C09147=1141.971,319.526,-76.453,-176.806,8.868,148.842
C09148=1141.967,319.774,-76.485,-176.803,8.872,148.842
C09149=1141.963,320.022,-76.518,-176.800,8.876,148.843
C09150=1141.958,320.270,-76.550,-176.798,8.880,148.843
C09151=1141.954,320.517,-76.583,-176.795,8.883,148.843
C09152=1141.950,320.766,-76.615,-176.792,8.887,148.843
C09153=1141.946,321.013,-76.648,-176.790,8.890,148.843
C09154=1141.942,321.261,-76.680,-176.787,8.894,148.844
C09155=1141.938,321.509,-76.713,-176.785,8.898,148.844
C09156=1141.934,321.757,-76.745,-176.782,8.902,148.844
C09157=1141.930,322.005,-76.778,-176.779,8.905,148.844
C09158=1141.926,322.253,-76.810,-176.776,8.909,148.844
C09159=1141.922,322.501,-76.843,-176.774,8.912,148.845
C09160=1141.917,322.748,-76.876,-176.771,8.916,148.845
C09161=1141.914,322.996,-76.908,-176.769,8.920,148.845
C09162=1141.910,323.243,-76.941,-176.766,8.924,148.845
C09163=1141.905,323.492,-76.973,-176.764,8.927,148.845
C09164=1141.901,323.739,-77.006,-176.761,8.931,148.846
C09165=1141.898,323.987,-77.039,-176.758,8.934,148.846
C09166=1141.893,324.235,-77.071,-176.756,8.938,148.846
C09167=1141.889,324.483,-77.105,-176.753,8.942,148.846
C09168=1141.886,324.730,-77.137,-176.751,8.945,148.847
C09169=1141.881,324.978,-77.170,-176.748,8.949,148.847
C09170=1141.877,325.226,-77.203,-176.746,8.953,148.847
C09171=1141.873,325.474,-77.236,-176.743,8.957,148.847
C09172=1141.869,325.722,-77.269,-176.741,8.960,148.848
C09173=1141.865,325.969,-77.302,-176.738,8.964,148.848
C09174=1141.861,326.218,-77.334,-176.735,8.967,148.848
C09175=1141.857,326.465,-77.367,-176.732,8.971,148.848
C09176=1141.853,326.713,-77.400,-176.730,8.975,148.848
C09177=1141.848,326.961,-77.434,-176.727,8.979,148.849
C09178=1141.844,327.209,-77.467,-176.724,8.983,148.849
C09179=1141.841,327.456,-77.499,-176.722,8.986,148.849
C09180=1141.836,327.704,-77.532,-176.719,8.990,148.849
C09181=1141.832,327.952,-77.565,-176.717,8.994,148.850
C09182=1141.828,328.200,-77.598,-176.714,8.998,148.850
C09183=1141.824,328.448,-77.631,-176.712,9.001,148.850
C09184=1141.820,328.695,-77.664,-176.709,9.005,148.850
C09185=1141.816,328.943,-77.698,-176.707,9.008,148.851
C09186=1141.812,329.191,-77.731,-176.704,9.012,148.851
C09187=1141.807,329.438,-77.764,-176.702,9.016,148.851
C09188=1141.804,329.687,-77.797,-176.699,9.020,148.851
C09189=1141.801,329.934,-77.830,-176.697,9.023,148.852
C09190=1141.796,330.182,-77.863,-176.694,9.027,148.852
C09191=1141.792,330.430,-77.896,-176.691,9.031,148.852
C09192=1141.788,330.677,-77.929,-176.688,9.035,148.852
C09193=1141.784,330.925,-77.963,-176.686,9.038,148.853
C09194=1141.780,331.173,-77.996,-176.683,9.042,148.853
C09195=1141.776,331.421,-78.029,-176.681,9.047,148.853
C09196=1141.772,331.668,-78.063,-176.678,9.050,148.853
C09197=1141.768,331.915,-78.096,-176.675,9.054,148.854
C09198=1141.764,332.164,-78.129,-176.673,9.057,148.854
C09199=1141.760,332.412,-78.163,-176.670,9.062,148.854
C09200=1141.755,332.660,-78.196,-176.668,9.065,148.854
C09201=1141.751,332.907,-78.229,-176.665,9.069,148.855
C09202=1141.747,333.155,-78.263,-176.663,9.072,148.855
C09203=1141.743,333.402,-78.296,-176.660,9.077,148.855
C09204=1141.739,333.650,-78.330,-176.657,9.081,148.856
C09205=1141.735,333.898,-78.363,-176.655,9.084,148.856
C09206=1141.732,334.146,-78.397,-176.652,9.088,148.856
C09207=1141.727,334.393,-78.430,-176.650,9.092,148.856
C09208=1141.723,334.641,-78.463,-176.647,9.096,148.857
C09209=1141.719,334.889,-78.497,-176.645,9.099,148.857
C09210=1141.716,335.137,-78.531,-176.642,9.103,148.857
C09211=1141.711,335.385,-78.564,-176.640,9.106,148.857
C09212=1141.707,335.632,-78.598,-176.637,9.111,148.858
C09213=1141.703,335.879,-78.632,-176.634,9.115,148.858
C09214=1141.699,336.127,-78.665,-176.632,9.118,148.858
C09215=1141.696,336.375,-78.699,-176.629,9.122,148.859
C09216=1141.691,336.623,-78.733,-176.627,9.126,148.859
C09217=1141.687,336.871,-78.766,-176.624,9.130,148.859
C09218=1141.683,337.118,-78.800,-176.621,9.134,148.859
C09219=1141.679,337.366,-78.833,-176.619,9.137,148.860
C09220=1141.676,337.613,-78.867,-176.616,9.141,148.860
C09221=1141.671,337.861,-78.901,-176.614,9.145,148.860
C09222=1141.667,338.109,-78.935,-176.612,9.149,148.860
C09223=1141.663,338.357,-78.968,-176.609,9.152,148.861
C09224=1141.659,338.604,-79.002,-176.606,9.156,148.861
C09225=1141.655,338.885,-79.041,-176.604,9.161,148.861
C09226=1141.650,339.165,-79.079,-176.601,9.165,148.862
C09227=1141.645,339.446,-79.118,-176.597,9.170,148.862
C09228=1141.641,339.726,-79.155,-176.595,9.174,148.862
C09229=1141.636,339.974,-79.189,-176.593,9.177,148.863
C09230=1141.633,340.222,-79.223,-176.590,9.181,148.863
C09231=1141.629,340.469,-79.257,-176.587,9.186,148.863
C09232=1141.624,340.717,-79.291,-176.585,9.189,148.863
C09233=1141.621,340.965,-79.325,-176.582,9.193,148.864
C09234=1141.617,341.212,-79.360,-176.579,9.198,148.864
C09235=1141.612,341.460,-79.393,-176.577,9.201,148.864
C09236=1141.609,341.708,-79.427,-176.574,9.205,148.865
C09237=1141.605,341.955,-79.462,-176.572,9.208,148.865
C09238=1141.601,342.203,-79.495,-176.569,9.213,148.865
C09239=1141.597,342.451,-79.530,-176.566,9.217,148.865
C09240=1141.593,342.698,-79.564,-176.564,9.220,148.866
C09241=1141.588,342.946,-79.598,-176.562,9.224,148.866
C09242=1141.585,343.194,-79.632,-176.559,9.229,148.867
C09243=1141.581,343.441,-79.665,-176.557,9.232,148.867
C09244=1141.576,343.689,-79.700,-176.554,9.236,148.867
C09245=1141.573,343.937,-79.734,-176.552,9.240,148.867
C09246=1141.568,344.184,-79.769,-176.549,9.244,148.868
C09247=1141.565,344.432,-79.803,-176.546,9.248,148.868
C09248=1141.561,344.679,-79.837,-176.544,9.251,148.868
C09249=1141.557,344.926,-79.871,-176.541,9.255,148.869
C09250=1141.553,345.174,-79.906,-176.539,9.260,148.869
C09251=1141.549,345.421,-79.940,-176.536,9.263,148.869
C09252=1141.545,345.670,-79.974,-176.534,9.267,148.870
C09253=1141.540,345.918,-80.008,-176.531,9.271,148.870
C09254=1141.537,346.165,-80.043,-176.529,9.275,148.870
C09255=1141.532,346.413,-80.077,-176.526,9.279,148.871
C09256=1141.529,346.660,-80.111,-176.524,9.282,148.871
C09257=1141.525,346.908,-80.146,-176.521,9.287,148.871
C09258=1141.521,347.155,-80.180,-176.518,9.291,148.871
C09259=1141.517,347.403,-80.215,-176.516,9.294,148.872
C09260=1141.512,347.650,-80.250,-176.513,9.299,148.872
C09261=1141.509,347.898,-80.284,-176.511,9.303,148.873
C09262=1141.505,348.145,-80.318,-176.509,9.306,148.873
C09263=1141.501,348.393,-80.353,-176.506,9.311,148.873
C09264=1141.497,348.641,-80.387,-176.503,9.315,148.873
C09265=1141.493,348.889,-80.422,-176.501,9.318,148.874
C09266=1141.489,349.136,-80.456,-176.498,9.322,148.874
C09267=1141.485,349.383,-80.491,-176.496,9.327,148.875
C09268=1141.481,349.631,-80.526,-176.494,9.330,148.875
C09269=1141.478,349.879,-80.560,-176.491,9.334,148.875
C09270=1141.473,350.126,-80.595,-176.488,9.338,148.876
C09271=1141.469,350.374,-80.629,-176.486,9.342,148.876
C09272=1141.465,350.621,-80.665,-176.483,9.346,148.876
C09273=1141.462,350.869,-80.699,-176.481,9.350,148.877
C09274=1141.458,351.117,-80.734,-176.478,9.354,148.877
C09275=1141.453,351.364,-80.769,-176.476,9.358,148.877
C09276=1141.449,351.612,-80.804,-176.473,9.362,148.878
C09277=1141.446,351.859,-80.837,-176.470,9.367,148.878
C09278=1141.442,352.106,-80.873,-176.468,9.370,148.878
C09279=1141.437,352.354,-80.908,-176.466,9.374,148.879
C09280=1141.433,352.602,-80.942,-176.463,9.378,148.879
C09281=1141.430,352.849,-80.977,-176.461,9.382,148.879
C09282=1141.426,353.097,-81.012,-176.458,9.386,148.880
C09283=1141.422,353.344,-81.047,-176.455,9.390,148.880
C09284=1141.418,353.591,-81.082,-176.453,9.394,148.880
C09285=1141.414,353.840,-81.117,-176.451,9.398,148.881
C09286=1141.410,354.087,-81.152,-176.448,9.402,148.881
C09287=1141.406,354.334,-81.186,-176.446,9.406,148.881
C09288=1141.402,354.582,-81.222,-176.443,9.410,148.882
C09289=1141.399,354.830,-81.256,-176.440,9.414,148.882
C09290=1141.394,355.077,-81.292,-176.438,9.418,148.882
C09291=1141.390,355.325,-81.326,-176.435,9.422,148.883
C09292=1141.387,355.572,-81.362,-176.433,9.426,148.883
C09293=1141.382,355.819,-81.397,-176.430,9.430,148.884
C09294=1141.378,356.067,-81.432,-176.428,9.434,148.884
C09295=1141.375,356.315,-81.468,-176.426,9.438,148.884
C09296=1141.371,356.562,-81.501,-176.423,9.442,148.885
C09297=1141.367,356.809,-81.537,-176.420,9.447,148.885
C09298=1141.364,357.057,-81.572,-176.418,9.450,148.885
C09299=1141.359,357.304,-81.607,-176.415,9.454,148.886
C09300=1141.355,357.552,-81.643,-176.413,9.459,148.886
C09301=1141.352,357.799,-81.678,-176.410,9.463,148.886
C09302=1141.347,358.047,-81.713,-176.408,9.466,148.887
C09303=1141.343,358.294,-81.748,-176.405,9.471,148.887
C09304=1141.340,358.542,-81.784,-176.402,9.475,148.887
C09305=1141.336,358.789,-81.819,-176.400,9.479,148.888
C09306=1141.332,359.037,-81.854,-176.398,9.483,148.888
C09307=1141.328,359.284,-81.889,-176.395,9.487,148.889
C09308=1141.324,359.532,-81.925,-176.393,9.491,148.889
C09309=1141.321,359.779,-81.960,-176.390,9.495,148.889
C09310=1141.316,360.026,-81.995,-176.388,9.499,148.890
C09311=1141.313,360.273,-82.031,-176.385,9.503,148.890
C09312=1141.309,360.521,-82.066,-176.382,9.507,148.890
C09313=1141.304,360.769,-82.102,-176.380,9.512,148.891
C09314=1141.301,361.017,-82.138,-176.377,9.516,148.891
C09315=1141.296,361.264,-82.173,-176.374,9.520,148.892
C09316=1141.293,361.511,-82.208,-176.372,9.524,148.892
C09317=1141.289,361.759,-82.244,-176.370,9.528,148.892
C09318=1141.285,362.006,-82.279,-176.367,9.532,148.893
C09319=1141.282,362.254,-82.315,-176.365,9.537,148.893
C09320=1141.277,362.500,-82.350,-176.362,9.541,148.893
C09321=1141.274,362.748,-82.386,-176.359,9.545,148.894
C09322=1141.269,362.996,-82.422,-176.356,9.549,148.894
C09323=1141.266,363.243,-82.457,-176.354,9.553,148.895
C09324=1141.262,363.491,-82.493,-176.352,9.557,148.895
C09325=1141.258,363.738,-82.528,-176.349,9.561,148.895
C09326=1141.255,363.986,-82.564,-176.346,9.565,148.896
C09327=1141.250,364.233,-82.600,-176.344,9.570,148.896
C09328=1141.246,364.480,-82.635,-176.341,9.574,148.897
C09329=1141.242,364.764,-82.676,-176.338,9.579,148.897
C09330=1141.238,365.048,-82.717,-176.335,9.583,148.898
C09331=1141.233,365.331,-82.759,-176.332,9.588,148.898
C09332=1141.229,365.616,-82.800,-176.329,9.594,148.898
C09333=1141.225,365.863,-82.835,-176.326,9.598,148.899
C09334=1141.221,366.109,-82.871,-176.323,9.602,148.899
C09335=1141.217,366.357,-82.907,-176.321,9.606,148.900
C09336=1141.213,366.604,-82.943,-176.319,9.610,148.900
C09337=1141.209,366.852,-82.978,-176.316,9.614,148.900
C09338=1141.205,367.099,-83.015,-176.313,9.618,148.901
C09339=1141.202,367.347,-83.051,-176.311,9.623,148.901
C09340=1141.198,367.594,-83.086,-176.308,9.627,148.901
C09341=1141.194,367.841,-83.123,-176.305,9.631,148.902
C09342=1141.190,368.089,-83.159,-176.303,9.636,148.902
C09343=1141.186,368.337,-83.195,-176.300,9.640,148.903
C09344=1141.183,368.584,-83.231,-176.297,9.644,148.903
C09345=1141.179,368.831,-83.267,-176.295,9.649,148.904
C09346=1141.174,369.079,-83.303,-176.292,9.653,148.904
C09347=1141.171,369.326,-83.339,-176.289,9.657,148.904
C09348=1141.167,369.574,-83.375,-176.287,9.661,148.905
C09349=1141.163,369.820,-83.412,-176.284,9.665,148.905
C09350=1141.160,370.068,-83.447,-176.281,9.670,148.905
C09351=1141.156,370.315,-83.484,-176.279,9.674,148.906
C09352=1141.152,370.563,-83.520,-176.276,9.678,148.906
C09353=1141.148,370.810,-83.556,-176.273,9.683,148.907
C09354=1141.144,371.057,-83.592,-176.271,9.687,148.907
C09355=1141.140,371.305,-83.629,-176.268,9.691,148.908
C09356=1141.136,371.552,-83.664,-176.266,9.695,148.908
C09357=1141.132,371.799,-83.701,-176.263,9.700,148.908
C09358=1141.129,372.046,-83.737,-176.261,9.704,148.909
C09359=1141.125,372.294,-83.774,-176.259,9.708,148.909
C09360=1141.121,372.541,-83.810,-176.256,9.712,148.910
C09361=1141.117,372.789,-83.846,-176.253,9.716,148.910
C09362=1141.113,373.036,-83.883,-176.251,9.721,148.910
C09363=1141.109,373.283,-83.919,-176.248,9.725,148.911
C09364=1141.105,373.530,-83.955,-176.246,9.729,148.911
C09365=1141.102,373.777,-83.992,-176.243,9.734,148.912
C09366=1141.098,374.025,-84.029,-176.241,9.737,148.912
C09367=1141.095,374.272,-84.065,-176.239,9.742,148.913
C09368=1141.090,374.520,-84.101,-176.236,9.746,148.913
C09369=1141.086,374.767,-84.138,-176.233,9.750,148.913
C09370=1141.083,375.014,-84.174,-176.231,9.754,148.914
C09371=1141.079,375.261,-84.211,-176.229,9.758,148.914
C09372=1141.075,375.508,-84.248,-176.226,9.763,148.915
C09373=1141.071,375.756,-84.284,-176.224,9.766,148.915
C09374=1141.067,376.003,-84.320,-176.222,9.770,148.916
C09375=1141.063,376.251,-84.358,-176.220,9.775,148.916
C09376=1141.060,376.498,-84.394,-176.218,9.779,148.917
C09377=1141.056,376.745,-84.431,-176.215,9.783,148.917
C09378=1141.052,376.992,-84.468,-176.213,9.787,148.918
C09379=1141.049,377.239,-84.504,-176.211,9.791,148.918
C09380=1141.044,377.486,-84.541,-176.209,9.795,148.919
C09381=1141.041,377.734,-84.578,-176.206,9.799,148.919
C09382=1141.037,377.982,-84.614,-176.205,9.803,148.920
C09383=1141.033,378.229,-84.650,-176.203,9.806,148.920
C09384=1141.029,378.476,-84.687,-176.200,9.811,148.920
C09385=1141.025,378.723,-84.724,-176.199,9.815,148.921
C09386=1141.021,378.970,-84.761,-176.197,9.818,148.921
C09387=1141.018,379.218,-84.798,-176.195,9.822,148.922
C09388=1141.014,379.465,-84.834,-176.194,9.826,148.923
C09389=1141.010,379.712,-84.872,-176.191,9.830,148.923
C09390=1141.006,379.959,-84.909,-176.189,9.834,148.924
C09391=1141.002,380.206,-84.946,-176.188,9.838,148.924
C09392=1140.999,380.454,-84.982,-176.186,9.841,148.925
C09393=1140.995,380.701,-85.019,-176.185,9.845,148.925
C09394=1140.991,380.948,-85.056,-176.183,9.848,148.926
C09395=1140.987,381.195,-85.093,-176.182,9.852,148.926
C09396=1140.984,381.443,-85.130,-176.180,9.856,148.927
C09397=1140.979,381.690,-85.167,-176.179,9.860,148.927
C09398=1140.976,381.937,-85.203,-176.177,9.862,148.928
C09399=1140.972,382.184,-85.241,-176.176,9.866,148.928
C09400=1140.969,382.432,-85.278,-176.175,9.869,148.929
C09401=1140.965,382.679,-85.315,-176.173,9.873,148.930
C09402=1140.961,382.926,-85.352,-176.172,9.876,148.930
C09403=1140.957,383.173,-85.389,-176.171,9.880,148.931
C09404=1140.953,383.421,-85.427,-176.170,9.884,148.931
C09405=1140.949,383.668,-85.463,-176.170,9.887,148.932
C09406=1140.945,383.915,-85.500,-176.169,9.890,148.933
C09407=1140.942,384.162,-85.537,-176.168,9.893,148.933
C09408=1140.939,384.409,-85.574,-176.167,9.896,148.934
C09409=1140.935,384.656,-85.611,-176.166,9.899,148.934
C09410=1140.930,384.904,-85.648,-176.166,9.903,148.935
C09411=1140.927,385.151,-85.685,-176.165,9.906,148.936
C09412=1140.923,385.398,-85.723,-176.165,9.908,148.936
C09413=1140.919,385.645,-85.760,-176.164,9.911,148.937
C09414=1140.916,385.893,-85.797,-176.164,9.915,148.938
C09415=1140.912,386.140,-85.834,-176.164,9.917,148.938
C09416=1140.908,386.387,-85.872,-176.163,9.921,148.939
C09417=1140.904,386.634,-85.908,-176.163,9.923,148.940
C09418=1140.900,386.882,-85.946,-176.163,9.925,148.940
C09419=1140.896,387.128,-85.983,-176.162,9.929,148.941
C09420=1140.892,387.376,-86.020,-176.162,9.931,148.942
C09421=1140.889,387.624,-86.057,-176.163,9.934,148.943
C09422=1140.886,387.870,-86.094,-176.163,9.936,148.943
C09423=1140.882,388.117,-86.131,-176.163,9.939,148.944
C09424=1140.878,388.365,-86.168,-176.163,9.942,148.945
C09425=1140.874,388.611,-86.206,-176.163,9.944,148.946
C09426=1140.870,388.859,-86.243,-176.163,9.947,148.946
C09427=1140.867,389.107,-86.280,-176.163,9.950,148.947
C09428=1140.863,389.353,-86.318,-176.164,9.952,148.948
C09429=1140.859,389.600,-86.354,-176.164,9.955,148.949
C09430=1140.856,389.848,-86.392,-176.165,9.957,148.949
C09431=1140.852,390.095,-86.429,-176.165,9.960,148.950
C09432=1140.847,390.342,-86.466,-176.165,9.962,148.951
C09433=1140.843,390.629,-86.510,-176.166,9.964,148.952
C09434=1140.839,390.917,-86.553,-176.167,9.967,148.952
C09435=1140.834,391.204,-86.596,-176.167,9.970,148.953
C09436=1140.830,391.491,-86.640,-176.168,9.973,148.954
C09437=1140.826,391.738,-86.677,-176.169,9.975,148.955
C09438=1140.823,391.985,-86.715,-176.169,9.978,148.956
C09439=1140.819,392.233,-86.751,-176.170,9.980,148.957
C09440=1140.815,392.480,-86.788,-176.171,9.982,148.957
C09441=1140.811,392.727,-86.826,-176.172,9.984,148.958
C09442=1140.807,392.974,-86.863,-176.173,9.987,148.959
C09443=1140.804,393.221,-86.901,-176.174,9.988,148.960
C09444=1140.800,393.469,-86.938,-176.174,9.991,148.961
C09445=1140.796,393.716,-86.975,-176.175,9.993,148.962
C09446=1140.792,393.962,-87.012,-176.176,9.995,148.962
C09447=1140.789,394.210,-87.050,-176.177,9.997,148.963
C09448=1140.785,394.457,-87.087,-176.178,9.999,148.964
C09449=1140.781,394.704,-87.124,-176.179,10.001,148.965
C09450=1140.777,394.952,-87.161,-176.180,10.004,148.966
C09451=1140.773,395.198,-87.199,-176.181,10.006,148.966
C09452=1140.769,395.446,-87.236,-176.182,10.008,148.967
C09453=1140.766,395.693,-87.274,-176.183,10.010,148.968
C09454=1140.762,395.940,-87.310,-176.184,10.012,148.969
C09455=1140.758,396.187,-87.347,-176.185,10.014,148.970
C09456=1140.755,396.435,-87.385,-176.186,10.016,148.971
C09457=1140.751,396.682,-87.422,-176.187,10.018,148.971
C09458=1140.747,396.928,-87.460,-176.188,10.021,148.972
C09459=1140.743,397.176,-87.497,-176.189,10.023,148.973
C09460=1140.739,397.423,-87.534,-176.190,10.025,148.974
C09461=1140.736,397.670,-87.571,-176.192,10.027,148.975
C09462=1140.732,397.918,-87.609,-176.193,10.029,148.976
C09463=1140.728,398.164,-87.646,-176.194,10.031,148.976
C09464=1140.724,398.412,-87.683,-176.195,10.032,148.977
C09465=1140.721,398.659,-87.721,-176.197,10.034,148.978
C09466=1140.717,398.906,-87.758,-176.198,10.037,148.979
C09467=1140.713,399.153,-87.795,-176.199,10.039,148.980
C09468=1140.710,399.401,-87.833,-176.200,10.041,148.981
C09469=1140.706,399.648,-87.869,-176.201,10.043,148.981
C09470=1140.702,399.894,-87.907,-176.202,10.045,148.982
C09471=1140.698,400.142,-87.944,-176.203,10.047,148.983
C09472=1140.694,400.389,-87.981,-176.205,10.048,148.984
C09473=1140.690,400.636,-88.019,-176.206,10.050,148.985
C09474=1140.687,400.884,-88.056,-176.208,10.053,148.986
C09475=1140.683,401.130,-88.093,-176.209,10.055,148.987
C09476=1140.679,401.378,-88.130,-176.210,10.057,148.987
C09477=1140.675,401.626,-88.168,-176.211,10.059,148.988
C09478=1140.672,401.872,-88.205,-176.212,10.061,148.989
C09479=1140.668,402.119,-88.242,-176.214,10.062,148.990
C09480=1140.664,402.367,-88.280,-176.215,10.064,148.991
C09481=1140.660,402.614,-88.317,-176.216,10.066,148.992
C09482=1140.656,402.861,-88.354,-176.217,10.069,148.993
C09483=1140.653,403.108,-88.392,-176.218,10.071,148.993
C09484=1140.649,403.355,-88.428,-176.219,10.073,148.994
C09485=1140.645,403.602,-88.466,-176.221,10.075,148.995
C09486=1140.642,403.850,-88.503,-176.222,10.076,148.996
C09487=1140.638,404.097,-88.540,-176.223,10.078,148.997
C09488=1140.634,404.344,-88.578,-176.225,10.080,148.998
C09489=1140.630,404.592,-88.615,-176.226,10.082,148.999
C09490=1140.627,404.838,-88.652,-176.227,10.085,148.999
C09491=1140.622,405.086,-88.690,-176.228,10.087,149.000
C09492=1140.618,405.333,-88.728,-176.229,10.089,149.001
C09493=1140.614,405.580,-88.765,-176.230,10.091,149.002
C09494=1140.610,405.827,-88.802,-176.231,10.093,149.003
C09495=1140.607,406.075,-88.840,-176.233,10.094,149.003
C09496=1140.603,406.322,-88.876,-176.234,10.096,149.004
C09497=1140.599,406.568,-88.914,-176.235,10.098,149.005
C09498=1140.596,406.816,-88.951,-176.237,10.101,149.006
C09499=1140.592,407.063,-88.988,-176.238,10.103,149.007
C09500=1140.588,407.310,-89.026,-176.239,10.105,149.008
C09501=1140.584,407.558,-89.063,-176.240,10.107,149.009
C09502=1140.581,407.804,-89.100,-176.241,10.109,149.009
C09503=1140.576,408.052,-89.137,-176.242,10.111,149.010
C09504=1140.573,408.299,-89.174,-176.243,10.113,149.011
C09505=1140.569,408.546,-89.212,-176.244,10.115,149.012
C09506=1140.565,408.793,-89.249,-176.245,10.117,149.013
C09507=1140.562,409.041,-89.287,-176.246,10.119,149.014
C09508=1140.558,409.288,-89.324,-176.247,10.121,149.014
C09509=1140.554,409.535,-89.361,-176.249,10.123,149.015
C09510=1140.551,409.782,-89.399,-176.250,10.125,149.016
C09511=1140.546,410.029,-89.435,-176.251,10.127,149.017
C09512=1140.543,410.276,-89.473,-176.252,10.129,149.018
C09513=1140.539,410.524,-89.510,-176.253,10.132,149.019
C09514=1140.535,410.771,-89.547,-176.254,10.134,149.019
C09515=1140.531,411.018,-89.585,-176.255,10.135,149.020
C09516=1140.528,411.265,-89.622,-176.255,10.138,149.021
C09517=1140.524,411.512,-89.659,-176.256,10.140,149.022
C09518=1140.520,411.759,-89.696,-176.257,10.142,149.023
C09519=1140.517,412.007,-89.734,-176.258,10.144,149.023
C09520=1140.513,412.254,-89.771,-176.259,10.147,149.024
C09521=1140.509,412.501,-89.808,-176.260,10.149,149.025
C09522=1140.505,412.748,-89.846,-176.261,10.151,149.026
C09523=1140.501,412.995,-89.883,-176.262,10.153,149.027
C09524=1140.497,413.242,-89.920,-176.263,10.155,149.027
C09525=1140.494,413.490,-89.958,-176.264,10.157,149.028
C09526=1140.490,413.736,-89.995,-176.265,10.159,149.029
C09527=1140.486,413.984,-90.032,-176.266,10.161,149.030
C09528=1140.483,414.231,-90.069,-176.266,10.164,149.031
C09529=1140.479,414.478,-90.107,-176.267,10.166,149.031
C09530=1140.475,414.726,-90.144,-176.268,10.168,149.032
C09531=1140.473,414.973,-90.181,-176.269,10.170,149.033
C09532=1140.471,415.220,-90.218,-176.270,10.172,149.034
C09533=1140.470,415.467,-90.255,-176.270,10.175,149.035
C09534=1140.469,415.714,-90.292,-176.271,10.177,149.035
C09535=1140.470,415.962,-90.329,-176.272,10.179,149.036
C09536=1140.470,416.209,-90.366,-176.273,10.181,149.037
C09537=1140.472,416.484,-90.407,-176.274,10.184,149.038
C09538=1140.475,416.759,-90.447,-176.275,10.186,149.039
C09539=1140.478,417.033,-90.488,-176.275,10.187,149.039
C09540=1140.482,417.308,-90.529,-176.276,10.190,149.040
C09541=1140.062,417.311,-90.579,-176.278,10.201,149.043
C09542=1140.057,417.033,-90.538,-176.277,10.199,149.043
C09543=1140.054,416.755,-90.497,-176.276,10.197,149.042
C09544=1140.052,416.476,-90.456,-176.276,10.194,149.041
C09545=1140.050,416.197,-90.415,-176.275,10.192,149.040
C09546=1140.049,415.949,-90.377,-176.273,10.190,149.039
C09547=1140.049,415.703,-90.341,-176.273,10.188,149.039
C09548=1140.050,415.455,-90.304,-176.272,10.185,149.038
C09549=1140.051,415.208,-90.267,-176.271,10.183,149.037
C09550=1140.053,414.961,-90.230,-176.271,10.181,149.036
C09551=1140.055,414.714,-90.193,-176.270,10.179,149.036
C09552=1140.059,414.466,-90.156,-176.269,10.176,149.035
C09553=1140.062,414.219,-90.118,-176.268,10.174,149.034
C09554=1140.066,413.972,-90.081,-176.267,10.173,149.033
C09555=1140.070,413.725,-90.043,-176.266,10.171,149.032
C09556=1140.073,413.478,-90.006,-176.265,10.169,149.032
C09557=1140.077,413.231,-89.968,-176.265,10.166,149.031
C09558=1140.081,412.984,-89.932,-176.264,10.164,149.030
C09559=1140.084,412.737,-89.894,-176.263,10.162,149.029
C09560=1140.088,412.489,-89.857,-176.261,10.159,149.028
C09561=1140.092,412.242,-89.820,-176.260,10.157,149.027
C09562=1140.096,411.995,-89.782,-176.260,10.156,149.027
C09563=1140.100,411.748,-89.745,-176.259,10.153,149.026
C09564=1140.104,411.501,-89.708,-176.258,10.151,149.025
C09565=1140.107,411.253,-89.670,-176.257,10.149,149.024
C09566=1140.111,411.007,-89.633,-176.256,10.147,149.023
C09567=1140.115,410.759,-89.596,-176.255,10.144,149.022
C09568=1140.118,410.512,-89.559,-176.254,10.142,149.022
C09569=1140.122,410.265,-89.521,-176.253,10.140,149.021
C09570=1140.126,410.018,-89.484,-176.252,10.138,149.020
C09571=1140.130,409.771,-89.446,-176.251,10.136,149.019
C09572=1140.134,409.523,-89.409,-176.250,10.134,149.018
C09573=1140.137,409.277,-89.372,-176.249,10.132,149.018
C09574=1140.141,409.029,-89.335,-176.247,10.130,149.017
C09575=1140.145,408.782,-89.298,-176.246,10.128,149.016
C09576=1140.149,408.535,-89.260,-176.245,10.126,149.015
C09577=1140.153,408.287,-89.222,-176.244,10.124,149.014
C09578=1140.157,408.040,-89.185,-176.243,10.122,149.013
C09579=1140.161,407.793,-89.148,-176.242,10.120,149.013
C09580=1140.164,407.545,-89.111,-176.241,10.118,149.012
C09581=1140.168,407.299,-89.073,-176.240,10.116,149.011
C09582=1140.172,407.052,-89.036,-176.238,10.113,149.010
C09583=1140.175,406.804,-88.998,-176.237,10.111,149.009
C09584=1140.180,406.557,-88.962,-176.236,10.109,149.008
C09585=1140.183,406.310,-88.924,-176.235,10.107,149.007
C09586=1140.187,406.063,-88.887,-176.234,10.105,149.007
C09587=1140.191,405.815,-88.850,-176.233,10.103,149.006
C09588=1140.195,405.569,-88.812,-176.232,10.101,149.005
C09589=1140.198,405.321,-88.775,-176.231,10.099,149.004
C09590=1140.202,405.074,-88.738,-176.229,10.096,149.003
C09591=1140.205,404.826,-88.700,-176.228,10.094,149.002
C09592=1140.209,404.580,-88.663,-176.227,10.093,149.001
C09593=1140.213,404.333,-88.626,-176.226,10.091,149.001
C09594=1140.217,404.085,-88.589,-176.224,10.089,149.000
C09595=1140.221,403.838,-88.551,-176.223,10.087,148.999
C09596=1140.225,403.591,-88.514,-176.222,10.085,148.998
C09597=1140.228,403.344,-88.476,-176.221,10.082,148.997
C09598=1140.232,403.097,-88.439,-176.220,10.080,148.996
C09599=1140.236,402.850,-88.402,-176.219,10.078,148.995
C09600=1140.239,402.602,-88.365,-176.217,10.077,148.995
C09601=1140.243,402.355,-88.328,-176.216,10.075,148.994
C09602=1140.247,402.108,-88.290,-176.215,10.073,148.993
C09603=1140.251,401.860,-88.253,-176.213,10.071,148.992
C09604=1140.254,401.614,-88.215,-176.212,10.068,148.991
C09605=1140.259,401.367,-88.179,-176.211,10.066,148.990
C09606=1140.262,401.119,-88.141,-176.210,10.064,148.990
C09607=1140.266,400.872,-88.104,-176.208,10.063,148.989
C09608=1140.270,400.625,-88.067,-176.207,10.061,148.988
C09609=1140.273,400.378,-88.029,-176.206,10.059,148.987
C09610=1140.277,400.131,-87.992,-176.205,10.057,148.986
C09611=1140.281,399.884,-87.955,-176.204,10.055,148.985
C09612=1140.284,399.636,-87.917,-176.203,10.052,148.984
C09613=1140.289,399.389,-87.880,-176.201,10.050,148.984
C09614=1140.292,399.142,-87.843,-176.200,10.049,148.983
C09615=1140.296,398.894,-87.806,-176.199,10.047,148.982
C09616=1140.300,398.648,-87.768,-176.198,10.045,148.981
C09617=1140.304,398.401,-87.731,-176.197,10.043,148.980
C09618=1140.307,398.153,-87.693,-176.195,10.041,148.979
C09619=1140.311,397.906,-87.656,-176.194,10.039,148.978
C09620=1140.315,397.659,-87.620,-176.193,10.036,148.978
C09621=1140.319,397.411,-87.581,-176.192,10.034,148.977
C09622=1140.323,397.164,-87.544,-176.191,10.032,148.976
C09623=1140.327,396.918,-87.507,-176.190,10.030,148.975
C09624=1140.330,396.670,-87.469,-176.188,10.028,148.974
C09625=1140.334,396.423,-87.432,-176.187,10.026,148.973
C09626=1140.338,396.176,-87.395,-176.186,10.024,148.973
C09627=1140.342,395.928,-87.358,-176.185,10.022,148.972
C09628=1140.346,395.682,-87.320,-176.184,10.020,148.971
C09629=1140.350,395.434,-87.283,-176.183,10.018,148.970
C09630=1140.353,395.187,-87.245,-176.182,10.016,148.969
C09631=1140.357,394.940,-87.208,-176.181,10.014,148.969
C09632=1140.361,394.693,-87.172,-176.180,10.012,148.968
C09633=1140.364,394.446,-87.134,-176.179,10.010,148.967
C09634=1140.368,394.198,-87.097,-176.178,10.008,148.966
C09635=1140.372,393.952,-87.059,-176.178,10.005,148.965
C09636=1140.376,393.704,-87.022,-176.176,10.003,148.964
C09637=1140.379,393.457,-86.984,-176.175,10.001,148.964
C09638=1140.384,393.210,-86.948,-176.175,9.999,148.963
C09639=1140.387,392.962,-86.910,-176.174,9.996,148.962
C09640=1140.391,392.716,-86.873,-176.173,9.994,148.961
C09641=1140.395,392.468,-86.836,-176.172,9.992,148.961
C09642=1140.398,392.221,-86.798,-176.172,9.990,148.960
C09643=1140.402,391.974,-86.761,-176.171,9.988,148.959
C09644=1140.406,391.726,-86.724,-176.170,9.986,148.958
C09645=1140.409,391.480,-86.686,-176.170,9.983,148.957
C09646=1140.414,391.192,-86.643,-176.169,9.980,148.956
C09647=1140.418,390.906,-86.600,-176.168,9.978,148.956
C09648=1140.423,390.618,-86.557,-176.168,9.975,148.955
C09649=1140.427,390.330,-86.513,-176.167,9.972,148.954
C09650=1140.431,390.083,-86.476,-176.167,9.969,148.953
C09651=1140.435,389.836,-86.439,-176.166,9.968,148.952
C09652=1140.438,389.589,-86.401,-176.166,9.965,148.952
C09653=1140.442,389.342,-86.364,-176.165,9.962,148.951
C09654=1140.446,389.095,-86.327,-176.165,9.960,148.950
C09655=1140.450,388.847,-86.289,-176.165,9.957,148.949
C09656=1140.454,388.600,-86.252,-176.164,9.955,148.949
C09657=1140.458,388.353,-86.216,-176.164,9.953,148.948
C09658=1140.460,388.106,-86.178,-176.164,9.950,148.947
C09659=1140.464,387.859,-86.141,-176.164,9.947,148.946
C09660=1140.468,387.612,-86.104,-176.164,9.944,148.946
C09661=1140.472,387.364,-86.067,-176.164,9.941,148.945
C09662=1140.476,387.117,-86.030,-176.164,9.939,148.944
C09663=1140.480,386.870,-85.993,-176.164,9.937,148.944
C09664=1140.483,386.623,-85.955,-176.165,9.933,148.943
C09665=1140.487,386.375,-85.918,-176.165,9.931,148.942
C09666=1140.491,386.128,-85.881,-176.165,9.928,148.942
C09667=1140.494,385.881,-85.843,-176.165,9.925,148.941
C09668=1140.498,385.634,-85.806,-176.166,9.922,148.940
C09669=1140.503,385.387,-85.770,-176.166,9.919,148.940
C09670=1140.506,385.139,-85.732,-176.167,9.916,148.939
C09671=1140.510,384.892,-85.695,-176.167,9.913,148.938
C09672=1140.514,384.645,-85.658,-176.168,9.910,148.938
C09673=1140.518,384.398,-85.621,-176.168,9.907,148.937
C09674=1140.521,384.151,-85.583,-176.169,9.904,148.937
C09675=1140.525,383.903,-85.546,-176.170,9.901,148.936
C09676=1140.529,383.656,-85.510,-176.171,9.898,148.935
C09677=1140.532,383.409,-85.473,-176.172,9.894,148.935
C09678=1140.536,383.162,-85.435,-176.173,9.891,148.934
C09679=1140.540,382.915,-85.398,-176.174,9.888,148.934
C09680=1140.544,382.668,-85.361,-176.176,9.884,148.933
C09681=1140.548,382.420,-85.324,-176.177,9.881,148.932
C09682=1140.551,382.173,-85.287,-176.177,9.877,148.932
C09683=1140.556,381.926,-85.250,-176.179,9.874,148.931
C09684=1140.559,381.679,-85.214,-176.181,9.870,148.931
C09685=1140.562,381.431,-85.176,-176.182,9.867,148.930
C09686=1140.566,381.184,-85.139,-176.183,9.863,148.930
C09687=1140.571,380.937,-85.103,-176.185,9.860,148.929
C09688=1140.575,380.690,-85.066,-176.187,9.856,148.929
C09689=1140.578,380.442,-85.028,-176.188,9.852,148.928
C09690=1140.582,380.195,-84.991,-176.190,9.848,148.928
C09691=1140.585,379.948,-84.955,-176.192,9.844,148.927
C09692=1140.589,379.701,-84.918,-176.194,9.841,148.927
C09693=1140.594,379.454,-84.881,-176.195,9.837,148.926
C09694=1140.597,379.206,-84.844,-176.197,9.833,148.925
C09695=1140.601,378.959,-84.807,-176.199,9.830,148.925
C09696=1140.604,378.712,-84.771,-176.201,9.826,148.924
C09697=1140.609,378.465,-84.734,-176.203,9.822,148.924
C09698=1140.613,378.218,-84.697,-176.205,9.818,148.924
C09699=1140.616,377.970,-84.660,-176.206,9.814,148.923
C09700=1140.619,377.723,-84.623,-176.209,9.810,148.922
C09701=1140.624,377.476,-84.587,-176.211,9.806,148.922
C09702=1140.628,377.228,-84.550,-176.213,9.802,148.922
C09703=1140.632,376.981,-84.513,-176.215,9.798,148.921
C09704=1140.635,376.734,-84.477,-176.218,9.794,148.921
C09705=1140.639,376.486,-84.440,-176.219,9.790,148.920
C09706=1140.643,376.239,-84.403,-176.222,9.786,148.920
C09707=1140.646,375.992,-84.367,-176.224,9.782,148.919
C09708=1140.650,375.745,-84.330,-176.226,9.778,148.919
C09709=1140.655,375.497,-84.293,-176.229,9.773,148.918
C09710=1140.658,375.250,-84.257,-176.231,9.770,148.918
C09711=1140.662,375.003,-84.220,-176.233,9.765,148.917
C09712=1140.666,374.755,-84.184,-176.236,9.761,148.917
C09713=1140.669,374.508,-84.147,-176.238,9.757,148.917
C09714=1140.673,374.261,-84.110,-176.241,9.753,148.916
C09715=1140.677,374.014,-84.074,-176.243,9.749,148.916
C09716=1140.681,373.766,-84.038,-176.246,9.744,148.915
C09717=1140.685,373.519,-84.001,-176.248,9.740,148.915
C09718=1140.688,373.272,-83.965,-176.250,9.737,148.914
C09719=1140.693,373.025,-83.928,-176.253,9.732,148.914
C09720=1140.696,372.777,-83.893,-176.255,9.728,148.914
C09721=1140.700,372.530,-83.856,-176.258,9.724,148.913
C09722=1140.704,372.283,-83.819,-176.261,9.719,148.913
C09723=1140.707,372.035,-83.783,-176.263,9.715,148.912
C09724=1140.712,371.787,-83.746,-176.266,9.711,148.912
C09725=1140.715,371.540,-83.710,-176.268,9.706,148.911
C09726=1140.719,371.293,-83.674,-176.271,9.703,148.911
C09727=1140.723,371.046,-83.637,-176.273,9.699,148.911
C09728=1140.727,370.798,-83.601,-176.276,9.694,148.910
C09729=1140.730,370.551,-83.565,-176.278,9.690,148.910
C09730=1140.735,370.303,-83.529,-176.281,9.686,148.910
C09731=1140.738,370.057,-83.493,-176.284,9.681,148.909
C09732=1140.742,369.809,-83.457,-176.286,9.677,148.909
C09733=1140.746,369.562,-83.420,-176.289,9.673,148.908
C09734=1140.750,369.314,-83.385,-176.292,9.668,148.908
C09735=1140.754,369.067,-83.348,-176.294,9.664,148.907
C09736=1140.757,368.820,-83.312,-176.297,9.660,148.907
C09737=1140.762,368.572,-83.276,-176.299,9.656,148.907
C09738=1140.765,368.325,-83.240,-176.302,9.651,148.906
C09739=1140.769,368.077,-83.204,-176.305,9.647,148.906
C09740=1140.773,367.830,-83.168,-176.307,9.643,148.905
C09741=1140.777,367.583,-83.132,-176.310,9.638,148.905
C09742=1140.782,367.336,-83.096,-176.312,9.634,148.905
C09743=1140.785,367.088,-83.060,-176.315,9.630,148.904
C09744=1140.789,366.841,-83.024,-176.318,9.626,148.904
C09745=1140.793,366.593,-82.988,-176.320,9.621,148.903
C09746=1140.797,366.346,-82.953,-176.323,9.617,148.903
C09747=1140.800,366.098,-82.917,-176.326,9.613,148.903
C09748=1140.804,365.851,-82.880,-176.328,9.608,148.902
C09749=1140.808,365.604,-82.845,-176.331,9.604,148.902
C09750=1140.812,365.320,-82.804,-176.334,9.600,148.901
C09751=1140.816,365.036,-82.763,-176.337,9.595,148.901
C09752=1140.821,364.753,-82.721,-176.340,9.590,148.901
C09753=1140.826,364.469,-82.680,-176.343,9.585,148.900
C09754=1140.830,364.222,-82.645,-176.345,9.581,148.900
C09755=1140.833,363.974,-82.609,-176.348,9.577,148.899
C09756=1140.838,363.726,-82.573,-176.351,9.573,148.899
C09757=1140.841,363.479,-82.538,-176.353,9.568,148.898
C09758=1140.845,363.231,-82.502,-176.356,9.564,148.898
C09759=1140.849,362.984,-82.467,-176.359,9.560,148.898
C09760=1140.853,362.737,-82.431,-176.361,9.555,148.897
C09761=1140.857,362.490,-82.396,-176.364,9.551,148.897
C09762=1140.861,362.242,-82.360,-176.367,9.547,148.897
C09763=1140.865,361.994,-82.324,-176.369,9.543,148.896
C09764=1140.868,361.747,-82.289,-176.372,9.539,148.896
C09765=1140.872,361.499,-82.253,-176.374,9.535,148.895
C09766=1140.876,361.253,-82.218,-176.377,9.531,148.895
C09767=1140.880,361.005,-82.182,-176.380,9.526,148.895
C09768=1140.883,360.758,-82.147,-176.382,9.522,148.894
C09769=1140.887,360.510,-82.111,-176.384,9.519,148.894
C09770=1140.891,360.263,-82.076,-176.387,9.514,148.894
C09771=1140.896,360.015,-82.040,-176.389,9.510,148.893
C09772=1140.900,359.767,-82.005,-176.392,9.506,148.893
C09773=1140.903,359.520,-81.970,-176.395,9.502,148.892
C09774=1140.907,359.272,-81.934,-176.397,9.497,148.892
C09775=1140.911,359.025,-81.899,-176.400,9.494,148.892
C09776=1140.915,358.778,-81.863,-176.402,9.490,148.891
C09777=1140.919,358.530,-81.828,-176.405,9.485,148.891
C09778=1140.923,358.282,-81.793,-176.408,9.481,148.891
C09779=1140.927,358.036,-81.758,-176.410,9.478,148.890
C09780=1140.931,357.788,-81.722,-176.413,9.473,148.890
C09781=1140.935,357.540,-81.687,-176.415,9.469,148.889
C09782=1140.938,357.292,-81.652,-176.418,9.465,148.889
C09783=1140.942,357.046,-81.617,-176.420,9.461,148.889
C09784=1140.946,356.798,-81.582,-176.422,9.457,148.888
C09785=1140.950,356.550,-81.546,-176.425,9.453,148.888
C09786=1140.954,356.304,-81.512,-176.428,9.449,148.888
C09787=1140.958,356.055,-81.477,-176.430,9.445,148.887
C09788=1140.961,355.808,-81.441,-176.433,9.441,148.887
C09789=1140.966,355.561,-81.406,-176.435,9.437,148.886
C09790=1140.970,355.313,-81.371,-176.438,9.433,148.886
C09791=1140.973,355.065,-81.336,-176.440,9.429,148.886
C09792=1140.978,354.818,-81.301,-176.443,9.424,148.885
C09793=1140.981,354.571,-81.266,-176.446,9.420,148.885
C09794=1140.985,354.322,-81.231,-176.447,9.417,148.885
C09795=1140.989,354.076,-81.196,-176.450,9.413,148.884
C09796=1140.993,353.828,-81.161,-176.453,9.408,148.884
C09797=1140.997,353.580,-81.126,-176.455,9.405,148.884
C09798=1141.001,353.333,-81.091,-176.458,9.401,148.883
C09799=1141.005,353.085,-81.056,-176.460,9.396,148.883
C09800=1141.009,352.838,-81.021,-176.463,9.392,148.883
C09801=1141.013,352.590,-80.987,-176.465,9.389,148.882
C09802=1141.016,352.343,-80.952,-176.468,9.385,148.882
C09803=1141.021,352.095,-80.917,-176.471,9.380,148.882
C09804=1141.025,351.847,-80.882,-176.473,9.377,148.881
C09805=1141.029,351.600,-80.847,-176.475,9.373,148.881
C09806=1141.032,351.353,-80.813,-176.478,9.369,148.881
C09807=1141.037,351.105,-80.778,-176.480,9.365,148.880
C09808=1141.041,350.858,-80.743,-176.483,9.361,148.880
C09809=1141.044,350.610,-80.709,-176.486,9.356,148.880
C09810=1141.048,350.362,-80.674,-176.488,9.353,148.879
C09811=1141.052,350.115,-80.639,-176.490,9.349,148.879
C09812=1141.057,349.867,-80.604,-176.493,9.344,148.878
C09813=1141.060,349.620,-80.570,-176.495,9.341,148.878
C09814=1141.064,349.372,-80.535,-176.498,9.337,148.878
C09815=1141.068,349.124,-80.501,-176.501,9.333,148.877
C09816=1141.072,348.878,-80.466,-176.503,9.328,148.877
C09817=1141.076,348.630,-80.431,-176.506,9.325,148.877
C09818=1141.080,348.382,-80.397,-176.509,9.321,148.877
C09819=1141.084,348.134,-80.363,-176.511,9.317,148.876
C09820=1141.088,347.887,-80.328,-176.513,9.313,148.876
C09821=1141.092,347.639,-80.293,-176.516,9.309,148.875
C09822=1141.096,347.392,-80.259,-176.519,9.305,148.875
C09823=1141.100,347.143,-80.225,-176.521,9.301,148.875
C09824=1141.104,346.896,-80.191,-176.524,9.297,148.875
C09825=1141.107,346.649,-80.155,-176.526,9.293,148.874
C09826=1141.112,346.401,-80.121,-176.528,9.290,148.874
C09827=1141.115,346.154,-80.086,-176.531,9.285,148.873
C09828=1141.120,345.906,-80.052,-176.533,9.282,148.873
C09829=1141.124,345.659,-80.018,-176.536,9.278,148.873
C09830=1141.128,345.411,-79.983,-176.539,9.273,148.873
C09831=1141.132,345.163,-79.950,-176.541,9.270,148.872
C09832=1141.136,344.915,-79.915,-176.544,9.266,148.872
C09833=1141.140,344.668,-79.881,-176.547,9.262,148.872
C09834=1141.144,344.420,-79.847,-176.548,9.258,148.871
C09835=1141.147,344.173,-79.813,-176.551,9.254,148.871
C09836=1141.152,343.925,-79.778,-176.554,9.250,148.871
C09837=1141.155,343.678,-79.744,-176.556,9.246,148.870
C09838=1141.160,343.430,-79.709,-176.559,9.242,148.870
C09839=1141.164,343.183,-79.676,-176.562,9.238,148.870
C09840=1141.168,342.934,-79.642,-176.564,9.235,148.869
C09841=1141.172,342.687,-79.608,-176.566,9.230,148.869
C09842=1141.176,342.439,-79.573,-176.569,9.227,148.869
C09843=1141.179,342.192,-79.539,-176.572,9.223,148.869
C09844=1141.184,341.944,-79.505,-176.574,9.219,148.868
C09845=1141.188,341.696,-79.471,-176.577,9.215,148.868
C09846=1141.191,341.449,-79.437,-176.579,9.211,148.868
C09847=1141.196,341.202,-79.403,-176.582,9.207,148.867
C09848=1141.200,340.953,-79.369,-176.584,9.204,148.867
C09849=1141.204,340.706,-79.335,-176.587,9.200,148.867
C09850=1141.208,340.459,-79.301,-176.589,9.196,148.866
C09851=1141.211,340.210,-79.267,-176.592,9.192,148.866
C09852=1141.216,339.963,-79.233,-176.595,9.188,148.866
C09853=1141.220,339.716,-79.199,-176.597,9.184,148.866
C09854=1141.225,339.435,-79.160,-176.600,9.180,148.865
C09855=1141.229,339.154,-79.122,-176.603,9.175,148.865
C09856=1141.233,338.874,-79.084,-176.606,9.171,148.865
C09857=1141.238,338.593,-79.046,-176.609,9.167,148.864
C09858=1141.242,338.345,-79.012,-176.611,9.162,148.864
C09859=1141.246,338.098,-78.978,-176.614,9.159,148.864
C09860=1141.250,337.850,-78.944,-176.617,9.155,148.863
C09861=1141.254,337.603,-78.910,-176.619,9.151,148.863
C09862=1141.258,337.354,-78.877,-176.621,9.147,148.863
C09863=1141.262,337.107,-78.843,-176.624,9.143,148.863
C09864=1141.266,336.859,-78.809,-176.627,9.140,148.862
C09865=1141.271,336.612,-78.776,-176.629,9.136,148.862
C09866=1141.274,336.364,-78.742,-176.631,9.132,148.862
C09867=1141.278,336.116,-78.709,-176.634,9.128,148.861
C09868=1141.282,335.869,-78.674,-176.637,9.124,148.861
C09869=1141.287,335.621,-78.641,-176.639,9.121,148.861
C09870=1141.290,335.372,-78.608,-176.642,9.117,148.861
C09871=1141.294,335.125,-78.574,-176.645,9.113,148.860
C09872=1141.298,334.878,-78.541,-176.647,9.109,148.860
C09873=1141.302,334.630,-78.507,-176.650,9.105,148.860
C09874=1141.306,334.383,-78.474,-176.652,9.102,148.859
C09875=1141.310,334.134,-78.439,-176.655,9.098,148.859
C09876=1141.314,333.886,-78.406,-176.657,9.094,148.859
C09877=1141.318,333.639,-78.372,-176.660,9.090,148.859
C09878=1141.322,333.391,-78.339,-176.662,9.087,148.858
C09879=1141.327,333.144,-78.306,-176.665,9.083,148.858
C09880=1141.331,332.896,-78.273,-176.668,9.078,148.858
C09881=1141.334,332.648,-78.239,-176.670,9.075,148.858
C09882=1141.338,332.400,-78.206,-176.673,9.071,148.857
C09883=1141.342,332.153,-78.172,-176.675,9.068,148.857
C09884=1141.346,331.905,-78.139,-176.678,9.064,148.857
C09885=1141.351,331.657,-78.106,-176.680,9.060,148.856
C09886=1141.355,331.410,-78.073,-176.683,9.056,148.856
C09887=1141.359,331.162,-78.040,-176.685,9.053,148.856
C09888=1141.363,330.914,-78.007,-176.688,9.049,148.856
C09889=1141.366,330.666,-77.972,-176.691,9.045,148.856
C09890=1141.370,330.419,-77.939,-176.693,9.041,148.855
C09891=1141.374,330.171,-77.906,-176.696,9.037,148.855
C09892=1141.379,329.923,-77.873,-176.699,9.034,148.855
C09893=1141.383,329.675,-77.840,-176.701,9.030,148.855
C09894=1141.387,329.428,-77.807,-176.704,9.026,148.854
C09895=1141.391,329.180,-77.773,-176.707,9.022,148.854
C09896=1141.395,328.932,-77.740,-176.709,9.019,148.854
C09897=1141.399,328.684,-77.707,-176.712,9.015,148.853
C09898=1141.403,328.437,-77.674,-176.714,9.011,148.853
C09899=1141.408,328.189,-77.641,-176.717,9.007,148.853
C09900=1141.412,327.941,-77.608,-176.719,9.004,148.853
C09901=1141.416,327.693,-77.575,-176.722,9.000,148.853
C09902=1141.420,327.445,-77.543,-176.724,8.997,148.852
C09903=1141.424,327.198,-77.510,-176.727,8.993,148.852
C09904=1141.428,326.950,-77.476,-176.729,8.989,148.852
C09905=1141.432,326.702,-77.443,-176.732,8.985,148.852
C09906=1141.435,326.454,-77.410,-176.734,8.982,148.851
C09907=1141.440,326.206,-77.377,-176.737,8.978,148.851
C09908=1141.443,325.958,-77.345,-176.740,8.973,148.851
C09909=1141.447,325.710,-77.312,-176.743,8.970,148.851
C09910=1141.452,325.463,-77.278,-176.746,8.966,148.850
C09911=1141.456,325.216,-77.246,-176.748,8.963,148.850
C09912=1141.461,324.967,-77.213,-176.751,8.959,148.850
C09913=1141.464,324.720,-77.181,-176.753,8.955,148.850
C09914=1141.468,324.472,-77.147,-176.756,8.951,148.849
C09915=1141.472,324.224,-77.114,-176.758,8.948,148.849
C09916=1141.477,323.976,-77.082,-176.761,8.944,148.849
C09917=1141.480,323.729,-77.049,-176.763,8.941,148.849
C09918=1141.484,323.481,-77.016,-176.766,8.936,148.849
C09919=1141.489,323.233,-76.984,-176.769,8.933,148.848
C09920=1141.492,322.985,-76.951,-176.771,8.929,148.848
C09921=1141.497,322.737,-76.919,-176.774,8.926,148.848
C09922=1141.501,322.489,-76.886,-176.777,8.922,148.848
C09923=1141.504,322.242,-76.853,-176.779,8.919,148.848
C09924=1141.509,321.993,-76.821,-176.781,8.915,148.847
C09925=1141.513,321.746,-76.787,-176.784,8.911,148.847
C09926=1141.517,321.498,-76.756,-176.787,8.908,148.847
C09927=1141.521,321.250,-76.722,-176.790,8.904,148.847
C09928=1141.526,321.002,-76.690,-176.792,8.901,148.847
C09929=1141.529,320.755,-76.658,-176.795,8.897,148.846
C09930=1141.534,320.506,-76.625,-176.797,8.893,148.846
C09931=1141.537,320.259,-76.593,-176.800,8.889,148.846
C09932=1141.541,320.011,-76.560,-176.802,8.886,148.846
C09933=1141.546,319.763,-76.527,-176.805,8.882,148.845
C09934=1141.549,319.515,-76.495,-176.808,8.879,148.845
C09935=1141.553,319.267,-76.462,-176.811,8.874,148.845
C09936=1141.558,319.020,-76.431,-176.813,8.871,148.845
C09937=1141.562,318.771,-76.398,-176.816,8.867,148.845
C09938=1141.566,318.524,-76.366,-176.818,8.864,148.844
C09939=1141.570,318.276,-76.333,-176.821,8.860,148.844
C09940=1141.574,318.028,-76.301,-176.824,8.857,148.844
C09941=1141.578,317.780,-76.268,-176.826,8.853,148.844
C09942=1141.582,317.533,-76.237,-176.829,8.849,148.844
C09943=1141.587,317.284,-76.204,-176.831,8.846,148.843
C09944=1141.590,317.037,-76.172,-176.834,8.842,148.843
C09945=1141.594,316.788,-76.139,-176.836,8.839,148.843
C09946=1141.598,316.540,-76.107,-176.839,8.835,148.843
C09947=1141.603,316.293,-76.075,-176.842,8.831,148.843
C09948=1141.607,316.045,-76.043,-176.845,8.827,148.842
C09949=1141.611,315.797,-76.010,-176.847,8.824,148.842
C09950=1141.615,315.549,-75.979,-176.849,8.821,148.842
C09951=1141.619,315.301,-75.946,-176.852,8.817,148.842
C09952=1141.623,315.053,-75.915,-176.855,8.814,148.842
C09953=1141.627,314.805,-75.883,-176.858,8.810,148.842
C09954=1141.631,314.557,-75.850,-176.860,8.806,148.841
C09955=1141.635,314.309,-75.818,-176.863,8.802,148.841
C09956=1141.639,314.062,-75.786,-176.865,8.799,148.841
C09957=1141.644,313.814,-75.754,-176.868,8.795,148.841
C09958=1141.648,313.536,-75.718,-176.871,8.792,148.841
C09959=1141.653,313.258,-75.682,-176.874,8.788,148.840
C09960=1141.657,312.981,-75.646,-176.877,8.784,148.840
C09961=1141.662,312.702,-75.611,-176.880,8.780,148.840
C09962=1141.667,312.454,-75.579,-176.883,8.776,148.840
C09963=1141.670,312.206,-75.547,-176.885,8.772,148.840
C09964=1141.675,311.958,-75.515,-176.888,8.768,148.840
C09965=1141.679,311.711,-75.483,-176.890,8.765,148.839
C09966=1141.683,311.463,-75.452,-176.893,8.762,148.839
C09967=1141.686,311.215,-75.420,-176.896,8.758,148.839
C09968=1141.691,310.967,-75.388,-176.898,8.755,148.839
C09969=1141.695,310.719,-75.356,-176.901,8.751,148.839
C09970=1141.699,310.471,-75.324,-176.904,8.747,148.839
C09971=1141.703,310.223,-75.292,-176.906,8.744,148.838
C09972=1141.708,309.975,-75.260,-176.909,8.740,148.838
C09973=1141.711,309.727,-75.228,-176.911,8.737,148.838
C09974=1141.716,309.479,-75.197,-176.914,8.733,148.838
C09975=1141.720,309.231,-75.166,-176.917,8.730,148.838
C09976=1141.725,308.983,-75.133,-176.919,8.727,148.838
C09977=1141.728,308.735,-75.102,-176.922,8.723,148.837
C09978=1141.732,308.487,-75.070,-176.925,8.719,148.837
C09979=1141.737,308.239,-75.039,-176.928,8.715,148.837
C09980=1141.740,307.991,-75.007,-176.930,8.712,148.837
C09981=1141.745,307.744,-74.976,-176.933,8.709,148.837
C09982=1141.749,307.496,-74.943,-176.936,8.705,148.837
C09983=1141.753,307.247,-74.912,-176.938,8.702,148.836
C09984=1141.758,307.000,-74.881,-176.941,8.698,148.836
C09985=1141.761,306.752,-74.849,-176.944,8.695,148.836
C09986=1141.766,306.504,-74.818,-176.946,8.691,148.836
C09987=1141.770,306.256,-74.786,-176.949,8.687,148.836
C09988=1141.774,306.008,-74.755,-176.951,8.684,148.836
C09989=1141.778,305.760,-74.724,-176.954,8.681,148.836
C09990=1141.782,305.512,-74.692,-176.957,8.677,148.836
C09991=1141.786,305.264,-74.661,-176.959,8.674,148.835
C09992=1141.791,305.016,-74.629,-176.962,8.670,148.835
C09993=1141.795,304.767,-74.598,-176.965,8.666,148.835
C09994=1141.800,304.520,-74.566,-176.967,8.664,148.835
C09995=1141.803,304.272,-74.534,-176.970,8.659,148.835
C09996=1141.808,304.024,-74.504,-176.973,8.656,148.835
//INST
///DATE 2021/06/25 14:31
///ATTR SC,RW,RJ
////FRAME ROBOT
///GROUP1 RB1
NOP
MOVL C00000 V=800.0 PL=0
MOVL C00001 V=800.0 PL=0
MOVL C00002 V=800.0 PL=0
MOVL C00003 V=800.0 PL=0
MOVL C00004 V=800.0 PL=0
MOVL C00005 V=800.0 PL=0
MOVL C00006 V=800.0 PL=0
MOVL C00007 V=800.0 PL=0
MOVL C00008 V=800.0 PL=0
MOVL C00009 V=800.0 PL=0
MOVL C00010 V=800.0 PL=0
MOVL C00011 V=800.0 PL=0
MOVL C00012 V=800.0 PL=0
MOVL C00013 V=800.0 PL=0
MOVL C00014 V=800.0 PL=0
MOVL C00015 V=800.0 PL=0
MOVL C00016 V=800.0 PL=0
MOVL C00017 V=800.0 PL=0
MOVL C00018 V=800.0 PL=0
MOVL C00019 V=800.0 PL=0
MOVL C00020 V=800.0 PL=0
MOVL C00021 V=800.0 PL=0
MOVL C00022 V=800.0 PL=0
MOVL C00023 V=800.0 PL=0
MOVL C00024 V=800.0 PL=0
MOVL C00025 V=800.0 PL=0
MOVL C00026 V=800.0 PL=0
MOVL C00027 V=800.0 PL=0
MOVL C00028 V=800.0 PL=0
MOVL C00029 V=800.0 PL=0
MOVL C00030 V=800.0 PL=0
MOVL C00031 V=800.0 PL=0
MOVL C00032 V=800.0 PL=0
MOVL C00033 V=800.0 PL=0
MOVL C00034 V=800.0 PL=0
MOVL C00035 V=800.0 PL=0
MOVL C00036 V=800.0 PL=0
MOVL C00037 V=800.0 PL=0
MOVL C00038 V=800.0 PL=0
MOVL C00039 V=800.0 PL=0
MOVL C00040 V=800.0 PL=0
MOVL C00041 V=800.0 PL=0
MOVL C00042 V=800.0 PL=0
MOVL C00043 V=800.0 PL=0
MOVL C00044 V=800.0 PL=0
MOVL C00045 V=800.0 PL=0
MOVL C00046 V=800.0 PL=0
MOVL C00047 V=800.0 PL=0
MOVL C00048 V=800.0 PL=0
MOVL C00049 V=800.0 PL=0
MOVL C00050 V=800.0 PL=0
MOVL C00051 V=800.0 PL=0
MOVL C00052 V=800.0 PL=0
MOVL C00053 V=800.0 PL=0
MOVL C00054 V=800.0 PL=0
MOVL C00055 V=800.0 PL=0
MOVL C00056 V=800.0 PL=0
MOVL C00057 V=800.0 PL=0
MOVL C00058 V=800.0 PL=0
MOVL C00059 V=800.0 PL=0
MOVL C00060 V=800.0 PL=0
MOVL C00061 V=800.0 PL=0
MOVL C00062 V=800.0 PL=0
MOVL C00063 V=800.0 PL=0
MOVL C00064 V=800.0 PL=0
MOVL C00065 V=800.0 PL=0
MOVL C00066 V=800.0 PL=0
MOVL C00067 V=800.0 PL=0
MOVL C00068 V=800.0 PL=0
MOVL C00069 V=800.0 PL=0
MOVL C00070 V=800.0 PL=0
MOVL C00071 V=800.0 PL=0
MOVL C00072 V=800.0 PL=0
MOVL C00073 V=800.0 PL=0
MOVL C00074 V=800.0 PL=0
MOVL C00075 V=800.0 PL=0
MOVL C00076 V=800.0 PL=0
MOVL C00077 V=800.0 PL=0
MOVL C00078 V=800.0 PL=0
MOVL C00079 V=800.0 PL=0
MOVL C00080 V=800.0 PL=0
MOVL C00081 V=800.0 PL=0
MOVL C00082 V=800.0 PL=0
MOVL C00083 V=800.0 PL=0
MOVL C00084 V=800.0 PL=0
MOVL C00085 V=800.0 PL=0
MOVL C00086 V=800.0 PL=0
MOVL C00087 V=800.0 PL=0
MOVL C00088 V=800.0 PL=0
MOVL C00089 V=800.0 PL=0
MOVL C00090 V=800.0 PL=0
MOVL C00091 V=800.0 PL=0
MOVL C00092 V=800.0 PL=0
MOVL C00093 V=800.0 PL=0
MOVL C00094 V=800.0 PL=0
MOVL C00095 V=800.0 PL=0
MOVL C00096 V=800.0 PL=0
MOVL C00097 V=800.0 PL=0
MOVL C00098 V=800.0 PL=0
MOVL C00099 V=800.0 PL=0
MOVL C00100 V=800.0 PL=0
MOVL C00101 V=800.0 PL=0
MOVL C00102 V=800.0 PL=0
MOVL C00103 V=800.0 PL=0
MOVL C00104 V=800.0 PL=0
MOVL C00105 V=800.0 PL=0
MOVL C00106 V=800.0 PL=0
MOVL C00107 V=800.0 PL=0
MOVL C00108 V=800.0 PL=0
MOVL C00109 V=800.0 PL=0
MOVL C00110 V=800.0 PL=0
MOVL C00111 V=800.0 PL=0
MOVL C00112 V=800.0 PL=0
MOVL C00113 V=800.0 PL=0
MOVL C00114 V=800.0 PL=0
MOVL C00115 V=800.0 PL=0
MOVL C00116 V=800.0 PL=0
MOVL C00117 V=800.0 PL=0
MOVL C00118 V=800.0 PL=0
MOVL C00119 V=800.0 PL=0
MOVL C00120 V=800.0 PL=0
MOVL C00121 V=800.0 PL=0
MOVL C00122 V=800.0 PL=0
MOVL C00123 V=800.0 PL=0
MOVL C00124 V=800.0 PL=0
MOVL C00125 V=800.0 PL=0
MOVL C00126 V=800.0 PL=0
MOVL C00127 V=800.0 PL=0
MOVL C00128 V=800.0 PL=0
MOVL C00129 V=800.0 PL=0
MOVL C00130 V=800.0 PL=0
MOVL C00131 V=800.0 PL=0
MOVL C00132 V=800.0 PL=0
MOVL C00133 V=800.0 PL=0
MOVL C00134 V=800.0 PL=0
MOVL C00135 V=800.0 PL=0
MOVL C00136 V=800.0 PL=0
MOVL C00137 V=800.0 PL=0
MOVL C00138 V=800.0 PL=0
MOVL C00139 V=800.0 PL=0
MOVL C00140 V=800.0 PL=0
MOVL C00141 V=800.0 PL=0
MOVL C00142 V=800.0 PL=0
MOVL C00143 V=800.0 PL=0
MOVL C00144 V=800.0 PL=0
MOVL C00145 V=800.0 PL=0
MOVL C00146 V=800.0 PL=0
MOVL C00147 V=800.0 PL=0
MOVL C00148 V=800.0 PL=0
MOVL C00149 V=800.0 PL=0
MOVL C00150 V=800.0 PL=0
MOVL C00151 V=800.0 PL=0
MOVL C00152 V=800.0 PL=0
MOVL C00153 V=800.0 PL=0
MOVL C00154 V=800.0 PL=0
MOVL C00155 V=800.0 PL=0
MOVL C00156 V=800.0 PL=0
MOVL C00157 V=800.0 PL=0
MOVL C00158 V=800.0 PL=0
MOVL C00159 V=800.0 PL=0
MOVL C00160 V=800.0 PL=0
MOVL C00161 V=800.0 PL=0
MOVL C00162 V=800.0 PL=0
MOVL C00163 V=800.0 PL=0
MOVL C00164 V=800.0 PL=0
MOVL C00165 V=800.0 PL=0
MOVL C00166 V=800.0 PL=0
MOVL C00167 V=800.0 PL=0
MOVL C00168 V=800.0 PL=0
MOVL C00169 V=800.0 PL=0
MOVL C00170 V=800.0 PL=0
MOVL C00171 V=800.0 PL=0
MOVL C00172 V=800.0 PL=0
MOVL C00173 V=800.0 PL=0
MOVL C00174 V=800.0 PL=0
MOVL C00175 V=800.0 PL=0
MOVL C00176 V=800.0 PL=0
MOVL C00177 V=800.0 PL=0
MOVL C00178 V=800.0 PL=0
MOVL C00179 V=800.0 PL=0
MOVL C00180 V=800.0 PL=0
MOVL C00181 V=800.0 PL=0
MOVL C00182 V=800.0 PL=0
MOVL C00183 V=800.0 PL=0
MOVL C00184 V=800.0 PL=0
MOVL C00185 V=800.0 PL=0
MOVL C00186 V=800.0 PL=0
MOVL C00187 V=800.0 PL=0
MOVL C00188 V=800.0 PL=0
MOVL C00189 V=800.0 PL=0
MOVL C00190 V=800.0 PL=0
MOVL C00191 V=800.0 PL=0
MOVL C00192 V=800.0 PL=0
MOVL C00193 V=800.0 PL=0
MOVL C00194 V=800.0 PL=0
MOVL C00195 V=800.0 PL=0
MOVL C00196 V=800.0 PL=0
MOVL C00197 V=800.0 PL=0
MOVL C00198 V=800.0 PL=0
MOVL C00199 V=800.0 PL=0
MOVL C00200 V=800.0 PL=0
MOVL C00201 V=800.0 PL=0
MOVL C00202 V=800.0 PL=0
MOVL C00203 V=800.0 PL=0
MOVL C00204 V=800.0 PL=0
MOVL C00205 V=800.0 PL=0
MOVL C00206 V=800.0 PL=0
MOVL C00207 V=800.0 PL=0
MOVL C00208 V=800.0 PL=0
MOVL C00209 V=800.0 PL=0
MOVL C00210 V=800.0 PL=0
MOVL C00211 V=800.0 PL=0
MOVL C00212 V=800.0 PL=0
MOVL C00213 V=800.0 PL=0
MOVL C00214 V=800.0 PL=0
MOVL C00215 V=800.0 PL=0
MOVL C00216 V=800.0 PL=0
MOVL C00217 V=800.0 PL=0
MOVL C00218 V=800.0 PL=0
MOVL C00219 V=800.0 PL=0
MOVL C00220 V=800.0 PL=0
MOVL C00221 V=800.0 PL=0
MOVL C00222 V=800.0 PL=0
MOVL C00223 V=800.0 PL=0
MOVL C00224 V=800.0 PL=0
MOVL C00225 V=800.0 PL=0
MOVL C00226 V=800.0 PL=0
MOVL C00227 V=800.0 PL=0
MOVL C00228 V=800.0 PL=0
MOVL C00229 V=800.0 PL=0
MOVL C00230 V=800.0 PL=0
MOVL C00231 V=800.0 PL=0
MOVL C00232 V=800.0 PL=0
MOVL C00233 V=800.0 PL=0
MOVL C00234 V=800.0 PL=0
MOVL C00235 V=800.0 PL=0
MOVL C00236 V=800.0 PL=0
MOVL C00237 V=800.0 PL=0
MOVL C00238 V=800.0 PL=0
MOVL C00239 V=800.0 PL=0
MOVL C00240 V=800.0 PL=0
MOVL C00241 V=800.0 PL=0
MOVL C00242 V=800.0 PL=0
MOVL C00243 V=800.0 PL=0
MOVL C00244 V=800.0 PL=0
MOVL C00245 V=800.0 PL=0
MOVL C00246 V=800.0 PL=0
MOVL C00247 V=800.0 PL=0
MOVL C00248 V=800.0 PL=0
MOVL C00249 V=800.0 PL=0
MOVL C00250 V=800.0 PL=0
MOVL C00251 V=800.0 PL=0
MOVL C00252 V=800.0 PL=0
MOVL C00253 V=800.0 PL=0
MOVL C00254 V=800.0 PL=0
MOVL C00255 V=800.0 PL=0
MOVL C00256 V=800.0 PL=0
MOVL C00257 V=800.0 PL=0
MOVL C00258 V=800.0 PL=0
MOVL C00259 V=800.0 PL=0
MOVL C00260 V=800.0 PL=0
MOVL C00261 V=800.0 PL=0
MOVL C00262 V=800.0 PL=0
MOVL C00263 V=800.0 PL=0
MOVL C00264 V=800.0 PL=0
MOVL C00265 V=800.0 PL=0
MOVL C00266 V=800.0 PL=0
MOVL C00267 V=800.0 PL=0
MOVL C00268 V=800.0 PL=0
MOVL C00269 V=800.0 PL=0
MOVL C00270 V=800.0 PL=0
MOVL C00271 V=800.0 PL=0
MOVL C00272 V=800.0 PL=0
MOVL C00273 V=800.0 PL=0
MOVL C00274 V=800.0 PL=0
MOVL C00275 V=800.0 PL=0
MOVL C00276 V=800.0 PL=0
MOVL C00277 V=800.0 PL=0
MOVL C00278 V=800.0 PL=0
MOVL C00279 V=800.0 PL=0
MOVL C00280 V=800.0 PL=0
MOVL C00281 V=800.0 PL=0
MOVL C00282 V=800.0 PL=0
MOVL C00283 V=800.0 PL=0
MOVL C00284 V=800.0 PL=0
MOVL C00285 V=800.0 PL=0
MOVL C00286 V=800.0 PL=0
MOVL C00287 V=800.0 PL=0
MOVL C00288 V=800.0 PL=0
MOVL C00289 V=800.0 PL=0
MOVL C00290 V=800.0 PL=0
MOVL C00291 V=800.0 PL=0
MOVL C00292 V=800.0 PL=0
MOVL C00293 V=800.0 PL=0
MOVL C00294 V=800.0 PL=0
MOVL C00295 V=800.0 PL=0
MOVL C00296 V=800.0 PL=0
MOVL C00297 V=800.0 PL=0
MOVL C00298 V=800.0 PL=0
MOVL C00299 V=800.0 PL=0
MOVL C00300 V=800.0 PL=0
MOVL C00301 V=800.0 PL=0
MOVL C00302 V=800.0 PL=0
MOVL C00303 V=800.0 PL=0
MOVL C00304 V=800.0 PL=0
MOVL C00305 V=800.0 PL=0
MOVL C00306 V=800.0 PL=0
MOVL C00307 V=800.0 PL=0
MOVL C00308 V=800.0 PL=0
MOVL C00309 V=800.0 PL=0
MOVL C00310 V=800.0 PL=0
MOVL C00311 V=800.0 PL=0
MOVL C00312 V=800.0 PL=0
MOVL C00313 V=800.0 PL=0
MOVL C00314 V=800.0 PL=0
MOVL C00315 V=800.0 PL=0
MOVL C00316 V=800.0 PL=0
MOVL C00317 V=800.0 PL=0
MOVL C00318 V=800.0 PL=0
MOVL C00319 V=800.0 PL=0
MOVL C00320 V=800.0 PL=0
MOVL C00321 V=800.0 PL=0
MOVL C00322 V=800.0 PL=0
MOVL C00323 V=800.0 PL=0
MOVL C00324 V=800.0 PL=0
MOVL C00325 V=800.0 PL=0
MOVL C00326 V=800.0 PL=0
MOVL C00327 V=800.0 PL=0
MOVL C00328 V=800.0 PL=0
MOVL C00329 V=800.0 PL=0
MOVL C00330 V=800.0 PL=0
MOVL C00331 V=800.0 PL=0
MOVL C00332 V=800.0 PL=0
MOVL C00333 V=800.0 PL=0
MOVL C00334 V=800.0 PL=0
MOVL C00335 V=800.0 PL=0
MOVL C00336 V=800.0 PL=0
MOVL C00337 V=800.0 PL=0
MOVL C00338 V=800.0 PL=0
MOVL C00339 V=800.0 PL=0
MOVL C00340 V=800.0 PL=0
MOVL C00341 V=800.0 PL=0
MOVL C00342 V=800.0 PL=0
MOVL C00343 V=800.0 PL=0
MOVL C00344 V=800.0 PL=0
MOVL C00345 V=800.0 PL=0
MOVL C00346 V=800.0 PL=0
MOVL C00347 V=800.0 PL=0
MOVL C00348 V=800.0 PL=0
MOVL C00349 V=800.0 PL=0
MOVL C00350 V=800.0 PL=0
MOVL C00351 V=800.0 PL=0
MOVL C00352 V=800.0 PL=0
MOVL C00353 V=800.0 PL=0
MOVL C00354 V=800.0 PL=0
MOVL C00355 V=800.0 PL=0
MOVL C00356 V=800.0 PL=0
MOVL C00357 V=800.0 PL=0
MOVL C00358 V=800.0 PL=0
MOVL C00359 V=800.0 PL=0
MOVL C00360 V=800.0 PL=0
MOVL C00361 V=800.0 PL=0
MOVL C00362 V=800.0 PL=0
MOVL C00363 V=800.0 PL=0
MOVL C00364 V=800.0 PL=0
MOVL C00365 V=800.0 PL=0
MOVL C00366 V=800.0 PL=0
MOVL C00367 V=800.0 PL=0
MOVL C00368 V=800.0 PL=0
MOVL C00369 V=800.0 PL=0
MOVL C00370 V=800.0 PL=0
MOVL C00371 V=800.0 PL=0
MOVL C00372 V=800.0 PL=0
MOVL C00373 V=800.0 PL=0
MOVL C00374 V=800.0 PL=0
MOVL C00375 V=800.0 PL=0
MOVL C00376 V=800.0 PL=0
MOVL C00377 V=800.0 PL=0
MOVL C00378 V=800.0 PL=0
MOVL C00379 V=800.0 PL=0
MOVL C00380 V=800.0 PL=0
MOVL C00381 V=800.0 PL=0
MOVL C00382 V=800.0 PL=0
MOVL C00383 V=800.0 PL=0
MOVL C00384 V=800.0 PL=0
MOVL C00385 V=800.0 PL=0
MOVL C00386 V=800.0 PL=0
MOVL C00387 V=800.0 PL=0
MOVL C00388 V=800.0 PL=0
MOVL C00389 V=800.0 PL=0
MOVL C00390 V=800.0 PL=0
MOVL C00391 V=800.0 PL=0
MOVL C00392 V=800.0 PL=0
MOVL C00393 V=800.0 PL=0
MOVL C00394 V=800.0 PL=0
MOVL C00395 V=800.0 PL=0
MOVL C00396 V=800.0 PL=0
MOVL C00397 V=800.0 PL=0
MOVL C00398 V=800.0 PL=0
MOVL C00399 V=800.0 PL=0
MOVL C00400 V=800.0 PL=0
MOVL C00401 V=800.0 PL=0
MOVL C00402 V=800.0 PL=0
MOVL C00403 V=800.0 PL=0
MOVL C00404 V=800.0 PL=0
MOVL C00405 V=800.0 PL=0
MOVL C00406 V=800.0 PL=0
MOVL C00407 V=800.0 PL=0
MOVL C00408 V=800.0 PL=0
MOVL C00409 V=800.0 PL=0
MOVL C00410 V=800.0 PL=0
MOVL C00411 V=800.0 PL=0
MOVL C00412 V=800.0 PL=0
MOVL C00413 V=800.0 PL=0
MOVL C00414 V=800.0 PL=0
MOVL C00415 V=800.0 PL=0
MOVL C00416 V=800.0 PL=0
MOVL C00417 V=800.0 PL=0
MOVL C00418 V=800.0 PL=0
MOVL C00419 V=800.0 PL=0
MOVL C00420 V=800.0 PL=0
MOVL C00421 V=800.0 PL=0
MOVL C00422 V=800.0 PL=0
MOVL C00423 V=800.0 PL=0
MOVL C00424 V=800.0 PL=0
MOVL C00425 V=800.0 PL=0
MOVL C00426 V=800.0 PL=0
MOVL C00427 V=800.0 PL=0
MOVL C00428 V=800.0 PL=0
MOVL C00429 V=800.0 PL=0
MOVL C00430 V=800.0 PL=0
MOVL C00431 V=800.0 PL=0
MOVL C00432 V=800.0 PL=0
MOVL C00433 V=800.0 PL=0
MOVL C00434 V=800.0 PL=0
MOVL C00435 V=800.0 PL=0
MOVL C00436 V=800.0 PL=0
MOVL C00437 V=800.0 PL=0
MOVL C00438 V=800.0 PL=0
MOVL C00439 V=800.0 PL=0
MOVL C00440 V=800.0 PL=0
MOVL C00441 V=800.0 PL=0
MOVL C00442 V=800.0 PL=0
MOVL C00443 V=800.0 PL=0
MOVL C00444 V=800.0 PL=0
MOVL C00445 V=800.0 PL=0
MOVL C00446 V=800.0 PL=0
MOVL C00447 V=800.0 PL=0
MOVL C00448 V=800.0 PL=0
MOVL C00449 V=800.0 PL=0
MOVL C00450 V=800.0 PL=0
MOVL C00451 V=800.0 PL=0
MOVL C00452 V=800.0 PL=0
MOVL C00453 V=800.0 PL=0
MOVL C00454 V=800.0 PL=0
MOVL C00455 V=800.0 PL=0
MOVL C00456 V=800.0 PL=0
MOVL C00457 V=800.0 PL=0
MOVL C00458 V=800.0 PL=0
MOVL C00459 V=800.0 PL=0
MOVL C00460 V=800.0 PL=0
MOVL C00461 V=800.0 PL=0
MOVL C00462 V=800.0 PL=0
MOVL C00463 V=800.0 PL=0
MOVL C00464 V=800.0 PL=0
MOVL C00465 V=800.0 PL=0
MOVL C00466 V=800.0 PL=0
MOVL C00467 V=800.0 PL=0
MOVL C00468 V=800.0 PL=0
MOVL C00469 V=800.0 PL=0
MOVL C00470 V=800.0 PL=0
MOVL C00471 V=800.0 PL=0
MOVL C00472 V=800.0 PL=0
MOVL C00473 V=800.0 PL=0
MOVL C00474 V=800.0 PL=0
MOVL C00475 V=800.0 PL=0
MOVL C00476 V=800.0 PL=0
MOVL C00477 V=800.0 PL=0
MOVL C00478 V=800.0 PL=0
MOVL C00479 V=800.0 PL=0
MOVL C00480 V=800.0 PL=0
MOVL C00481 V=800.0 PL=0
MOVL C00482 V=800.0 PL=0
MOVL C00483 V=800.0 PL=0
MOVL C00484 V=800.0 PL=0
MOVL C00485 V=800.0 PL=0
MOVL C00486 V=800.0 PL=0
MOVL C00487 V=800.0 PL=0
MOVL C00488 V=800.0 PL=0
MOVL C00489 V=800.0 PL=0
MOVL C00490 V=800.0 PL=0
MOVL C00491 V=800.0 PL=0
MOVL C00492 V=800.0 PL=0
MOVL C00493 V=800.0 PL=0
MOVL C00494 V=800.0 PL=0
MOVL C00495 V=800.0 PL=0
MOVL C00496 V=800.0 PL=0
MOVL C00497 V=800.0 PL=0
MOVL C00498 V=800.0 PL=0
MOVL C00499 V=800.0 PL=0
MOVL C00500 V=800.0 PL=0
MOVL C00501 V=800.0 PL=0
MOVL C00502 V=800.0 PL=0
MOVL C00503 V=800.0 PL=0
MOVL C00504 V=800.0 PL=0
MOVL C00505 V=800.0 PL=0
MOVL C00506 V=800.0 PL=0
MOVL C00507 V=800.0 PL=0
MOVL C00508 V=800.0 PL=0
MOVL C00509 V=800.0 PL=0
MOVL C00510 V=800.0 PL=0
MOVL C00511 V=800.0 PL=0
MOVL C00512 V=800.0 PL=0
MOVL C00513 V=800.0 PL=0
MOVL C00514 V=800.0 PL=0
MOVL C00515 V=800.0 PL=0
MOVL C00516 V=800.0 PL=0
MOVL C00517 V=800.0 PL=0
MOVL C00518 V=800.0 PL=0
MOVL C00519 V=800.0 PL=0
MOVL C00520 V=800.0 PL=0
MOVL C00521 V=800.0 PL=0
MOVL C00522 V=800.0 PL=0
MOVL C00523 V=800.0 PL=0
MOVL C00524 V=800.0 PL=0
MOVL C00525 V=800.0 PL=0
MOVL C00526 V=800.0 PL=0
MOVL C00527 V=800.0 PL=0
MOVL C00528 V=800.0 PL=0
MOVL C00529 V=800.0 PL=0
MOVL C00530 V=800.0 PL=0
MOVL C00531 V=800.0 PL=0
MOVL C00532 V=800.0 PL=0
MOVL C00533 V=800.0 PL=0
MOVL C00534 V=800.0 PL=0
MOVL C00535 V=800.0 PL=0
MOVL C00536 V=800.0 PL=0
MOVL C00537 V=800.0 PL=0
MOVL C00538 V=800.0 PL=0
MOVL C00539 V=800.0 PL=0
MOVL C00540 V=800.0 PL=0
MOVL C00541 V=800.0 PL=0
MOVL C00542 V=800.0 PL=0
MOVL C00543 V=800.0 PL=0
MOVL C00544 V=800.0 PL=0
MOVL C00545 V=800.0 PL=0
MOVL C00546 V=800.0 PL=0
MOVL C00547 V=800.0 PL=0
MOVL C00548 V=800.0 PL=0
MOVL C00549 V=800.0 PL=0
MOVL C00550 V=800.0 PL=0
MOVL C00551 V=800.0 PL=0
MOVL C00552 V=800.0 PL=0
MOVL C00553 V=800.0 PL=0
MOVL C00554 V=800.0 PL=0
MOVL C00555 V=800.0 PL=0
MOVL C00556 V=800.0 PL=0
MOVL C00557 V=800.0 PL=0
MOVL C00558 V=800.0 PL=0
MOVL C00559 V=800.0 PL=0
MOVL C00560 V=800.0 PL=0
MOVL C00561 V=800.0 PL=0
MOVL C00562 V=800.0 PL=0
MOVL C00563 V=800.0 PL=0
MOVL C00564 V=800.0 PL=0
MOVL C00565 V=800.0 PL=0
MOVL C00566 V=800.0 PL=0
MOVL C00567 V=800.0 PL=0
MOVL C00568 V=800.0 PL=0
MOVL C00569 V=800.0 PL=0
MOVL C00570 V=800.0 PL=0
MOVL C00571 V=800.0 PL=0
MOVL C00572 V=800.0 PL=0
MOVL C00573 V=800.0 PL=0
MOVL C00574 V=800.0 PL=0
MOVL C00575 V=800.0 PL=0
MOVL C00576 V=800.0 PL=0
MOVL C00577 V=800.0 PL=0
MOVL C00578 V=800.0 PL=0
MOVL C00579 V=800.0 PL=0
MOVL C00580 V=800.0 PL=0
MOVL C00581 V=800.0 PL=0
MOVL C00582 V=800.0 PL=0
MOVL C00583 V=800.0 PL=0
MOVL C00584 V=800.0 PL=0
MOVL C00585 V=800.0 PL=0
MOVL C00586 V=800.0 PL=0
MOVL C00587 V=800.0 PL=0
MOVL C00588 V=800.0 PL=0
MOVL C00589 V=800.0 PL=0
MOVL C00590 V=800.0 PL=0
MOVL C00591 V=800.0 PL=0
MOVL C00592 V=800.0 PL=0
MOVL C00593 V=800.0 PL=0
MOVL C00594 V=800.0 PL=0
MOVL C00595 V=800.0 PL=0
MOVL C00596 V=800.0 PL=0
MOVL C00597 V=800.0 PL=0
MOVL C00598 V=800.0 PL=0
MOVL C00599 V=800.0 PL=0
MOVL C00600 V=800.0 PL=0
MOVL C00601 V=800.0 PL=0
MOVL C00602 V=800.0 PL=0
MOVL C00603 V=800.0 PL=0
MOVL C00604 V=800.0 PL=0
MOVL C00605 V=800.0 PL=0
MOVL C00606 V=800.0 PL=0
MOVL C00607 V=800.0 PL=0
MOVL C00608 V=800.0 PL=0
MOVL C00609 V=800.0 PL=0
MOVL C00610 V=800.0 PL=0
MOVL C00611 V=800.0 PL=0
MOVL C00612 V=800.0 PL=0
MOVL C00613 V=800.0 PL=0
MOVL C00614 V=800.0 PL=0
MOVL C00615 V=800.0 PL=0
MOVL C00616 V=800.0 PL=0
MOVL C00617 V=800.0 PL=0
MOVL C00618 V=800.0 PL=0
MOVL C00619 V=800.0 PL=0
MOVL C00620 V=800.0 PL=0
MOVL C00621 V=800.0 PL=0
MOVL C00622 V=800.0 PL=0
MOVL C00623 V=800.0 PL=0
MOVL C00624 V=800.0 PL=0
MOVL C00625 V=800.0 PL=0
MOVL C00626 V=800.0 PL=0
MOVL C00627 V=800.0 PL=0
MOVL C00628 V=800.0 PL=0
MOVL C00629 V=800.0 PL=0
MOVL C00630 V=800.0 PL=0
MOVL C00631 V=800.0 PL=0
MOVL C00632 V=800.0 PL=0
MOVL C00633 V=800.0 PL=0
MOVL C00634 V=800.0 PL=0
MOVL C00635 V=800.0 PL=0
MOVL C00636 V=800.0 PL=0
MOVL C00637 V=800.0 PL=0
MOVL C00638 V=800.0 PL=0
MOVL C00639 V=800.0 PL=0
MOVL C00640 V=800.0 PL=0
MOVL C00641 V=800.0 PL=0
MOVL C00642 V=800.0 PL=0
MOVL C00643 V=800.0 PL=0
MOVL C00644 V=800.0 PL=0
MOVL C00645 V=800.0 PL=0
MOVL C00646 V=800.0 PL=0
MOVL C00647 V=800.0 PL=0
MOVL C00648 V=800.0 PL=0
MOVL C00649 V=800.0 PL=0
MOVL C00650 V=800.0 PL=0
MOVL C00651 V=800.0 PL=0
MOVL C00652 V=800.0 PL=0
MOVL C00653 V=800.0 PL=0
MOVL C00654 V=800.0 PL=0
MOVL C00655 V=800.0 PL=0
MOVL C00656 V=800.0 PL=0
MOVL C00657 V=800.0 PL=0
MOVL C00658 V=800.0 PL=0
MOVL C00659 V=800.0 PL=0
MOVL C00660 V=800.0 PL=0
MOVL C00661 V=800.0 PL=0
MOVL C00662 V=800.0 PL=0
MOVL C00663 V=800.0 PL=0
MOVL C00664 V=800.0 PL=0
MOVL C00665 V=800.0 PL=0
MOVL C00666 V=800.0 PL=0
MOVL C00667 V=800.0 PL=0
MOVL C00668 V=800.0 PL=0
MOVL C00669 V=800.0 PL=0
MOVL C00670 V=800.0 PL=0
MOVL C00671 V=800.0 PL=0
MOVL C00672 V=800.0 PL=0
MOVL C00673 V=800.0 PL=0
MOVL C00674 V=800.0 PL=0
MOVL C00675 V=800.0 PL=0
MOVL C00676 V=800.0 PL=0
MOVL C00677 V=800.0 PL=0
MOVL C00678 V=800.0 PL=0
MOVL C00679 V=800.0 PL=0
MOVL C00680 V=800.0 PL=0
MOVL C00681 V=800.0 PL=0
MOVL C00682 V=800.0 PL=0
MOVL C00683 V=800.0 PL=0
MOVL C00684 V=800.0 PL=0
MOVL C00685 V=800.0 PL=0
MOVL C00686 V=800.0 PL=0
MOVL C00687 V=800.0 PL=0
MOVL C00688 V=800.0 PL=0
MOVL C00689 V=800.0 PL=0
MOVL C00690 V=800.0 PL=0
MOVL C00691 V=800.0 PL=0
MOVL C00692 V=800.0 PL=0
MOVL C00693 V=800.0 PL=0
MOVL C00694 V=800.0 PL=0
MOVL C00695 V=800.0 PL=0
MOVL C00696 V=800.0 PL=0
MOVL C00697 V=800.0 PL=0
MOVL C00698 V=800.0 PL=0
MOVL C00699 V=800.0 PL=0
MOVL C00700 V=800.0 PL=0
MOVL C00701 V=800.0 PL=0
MOVL C00702 V=800.0 PL=0
MOVL C00703 V=800.0 PL=0
MOVL C00704 V=800.0 PL=0
MOVL C00705 V=800.0 PL=0
MOVL C00706 V=800.0 PL=0
MOVL C00707 V=800.0 PL=0
MOVL C00708 V=800.0 PL=0
MOVL C00709 V=800.0 PL=0
MOVL C00710 V=800.0 PL=0
MOVL C00711 V=800.0 PL=0
MOVL C00712 V=800.0 PL=0
MOVL C00713 V=800.0 PL=0
MOVL C00714 V=800.0 PL=0
MOVL C00715 V=800.0 PL=0
MOVL C00716 V=800.0 PL=0
MOVL C00717 V=800.0 PL=0
MOVL C00718 V=800.0 PL=0
MOVL C00719 V=800.0 PL=0
MOVL C00720 V=800.0 PL=0
MOVL C00721 V=800.0 PL=0
MOVL C00722 V=800.0 PL=0
MOVL C00723 V=800.0 PL=0
MOVL C00724 V=800.0 PL=0
MOVL C00725 V=800.0 PL=0
MOVL C00726 V=800.0 PL=0
MOVL C00727 V=800.0 PL=0
MOVL C00728 V=800.0 PL=0
MOVL C00729 V=800.0 PL=0
MOVL C00730 V=800.0 PL=0
MOVL C00731 V=800.0 PL=0
MOVL C00732 V=800.0 PL=0
MOVL C00733 V=800.0 PL=0
MOVL C00734 V=800.0 PL=0
MOVL C00735 V=800.0 PL=0
MOVL C00736 V=800.0 PL=0
MOVL C00737 V=800.0 PL=0
MOVL C00738 V=800.0 PL=0
MOVL C00739 V=800.0 PL=0
MOVL C00740 V=800.0 PL=0
MOVL C00741 V=800.0 PL=0
MOVL C00742 V=800.0 PL=0
MOVL C00743 V=800.0 PL=0
MOVL C00744 V=800.0 PL=0
MOVL C00745 V=800.0 PL=0
MOVL C00746 V=800.0 PL=0
MOVL C00747 V=800.0 PL=0
MOVL C00748 V=800.0 PL=0
MOVL C00749 V=800.0 PL=0
MOVL C00750 V=800.0 PL=0
MOVL C00751 V=800.0 PL=0
MOVL C00752 V=800.0 PL=0
MOVL C00753 V=800.0 PL=0
MOVL C00754 V=800.0 PL=0
MOVL C00755 V=800.0 PL=0
MOVL C00756 V=800.0 PL=0
MOVL C00757 V=800.0 PL=0
MOVL C00758 V=800.0 PL=0
MOVL C00759 V=800.0 PL=0
MOVL C00760 V=800.0 PL=0
MOVL C00761 V=800.0 PL=0
MOVL C00762 V=800.0 PL=0
MOVL C00763 V=800.0 PL=0
MOVL C00764 V=800.0 PL=0
MOVL C00765 V=800.0 PL=0
MOVL C00766 V=800.0 PL=0
MOVL C00767 V=800.0 PL=0
MOVL C00768 V=800.0 PL=0
MOVL C00769 V=800.0 PL=0
MOVL C00770 V=800.0 PL=0
MOVL C00771 V=800.0 PL=0
MOVL C00772 V=800.0 PL=0
MOVL C00773 V=800.0 PL=0
MOVL C00774 V=800.0 PL=0
MOVL C00775 V=800.0 PL=0
MOVL C00776 V=800.0 PL=0
MOVL C00777 V=800.0 PL=0
MOVL C00778 V=800.0 PL=0
MOVL C00779 V=800.0 PL=0
MOVL C00780 V=800.0 PL=0
MOVL C00781 V=800.0 PL=0
MOVL C00782 V=800.0 PL=0
MOVL C00783 V=800.0 PL=0
MOVL C00784 V=800.0 PL=0
MOVL C00785 V=800.0 PL=0
MOVL C00786 V=800.0 PL=0
MOVL C00787 V=800.0 PL=0
MOVL C00788 V=800.0 PL=0
MOVL C00789 V=800.0 PL=0
MOVL C00790 V=800.0 PL=0
MOVL C00791 V=800.0 PL=0
MOVL C00792 V=800.0 PL=0
MOVL C00793 V=800.0 PL=0
MOVL C00794 V=800.0 PL=0
MOVL C00795 V=800.0 PL=0
MOVL C00796 V=800.0 PL=0
MOVL C00797 V=800.0 PL=0
MOVL C00798 V=800.0 PL=0
MOVL C00799 V=800.0 PL=0
MOVL C00800 V=800.0 PL=0
MOVL C00801 V=800.0 PL=0
MOVL C00802 V=800.0 PL=0
MOVL C00803 V=800.0 PL=0
MOVL C00804 V=800.0 PL=0
MOVL C00805 V=800.0 PL=0
MOVL C00806 V=800.0 PL=0
MOVL C00807 V=800.0 PL=0
MOVL C00808 V=800.0 PL=0
MOVL C00809 V=800.0 PL=0
MOVL C00810 V=800.0 PL=0
MOVL C00811 V=800.0 PL=0
MOVL C00812 V=800.0 PL=0
MOVL C00813 V=800.0 PL=0
MOVL C00814 V=800.0 PL=0
MOVL C00815 V=800.0 PL=0
MOVL C00816 V=800.0 PL=0
MOVL C00817 V=800.0 PL=0
MOVL C00818 V=800.0 PL=0
MOVL C00819 V=800.0 PL=0
MOVL C00820 V=800.0 PL=0
MOVL C00821 V=800.0 PL=0
MOVL C00822 V=800.0 PL=0
MOVL C00823 V=800.0 PL=0
MOVL C00824 V=800.0 PL=0
MOVL C00825 V=800.0 PL=0
MOVL C00826 V=800.0 PL=0
MOVL C00827 V=800.0 PL=0
MOVL C00828 V=800.0 PL=0
MOVL C00829 V=800.0 PL=0
MOVL C00830 V=800.0 PL=0
MOVL C00831 V=800.0 PL=0
MOVL C00832 V=800.0 PL=0
MOVL C00833 V=800.0 PL=0
MOVL C00834 V=800.0 PL=0
MOVL C00835 V=800.0 PL=0
MOVL C00836 V=800.0 PL=0
MOVL C00837 V=800.0 PL=0
MOVL C00838 V=800.0 PL=0
MOVL C00839 V=800.0 PL=0
MOVL C00840 V=800.0 PL=0
MOVL C00841 V=800.0 PL=0
MOVL C00842 V=800.0 PL=0
MOVL C00843 V=800.0 PL=0
MOVL C00844 V=800.0 PL=0
MOVL C00845 V=800.0 PL=0
MOVL C00846 V=800.0 PL=0
MOVL C00847 V=800.0 PL=0
MOVL C00848 V=800.0 PL=0
MOVL C00849 V=800.0 PL=0
MOVL C00850 V=800.0 PL=0
MOVL C00851 V=800.0 PL=0
MOVL C00852 V=800.0 PL=0
MOVL C00853 V=800.0 PL=0
MOVL C00854 V=800.0 PL=0
MOVL C00855 V=800.0 PL=0
MOVL C00856 V=800.0 PL=0
MOVL C00857 V=800.0 PL=0
MOVL C00858 V=800.0 PL=0
MOVL C00859 V=800.0 PL=0
MOVL C00860 V=800.0 PL=0
MOVL C00861 V=800.0 PL=0
MOVL C00862 V=800.0 PL=0
MOVL C00863 V=800.0 PL=0
MOVL C00864 V=800.0 PL=0
MOVL C00865 V=800.0 PL=0
MOVL C00866 V=800.0 PL=0
MOVL C00867 V=800.0 PL=0
MOVL C00868 V=800.0 PL=0
MOVL C00869 V=800.0 PL=0
MOVL C00870 V=800.0 PL=0
MOVL C00871 V=800.0 PL=0
MOVL C00872 V=800.0 PL=0
MOVL C00873 V=800.0 PL=0
MOVL C00874 V=800.0 PL=0
MOVL C00875 V=800.0 PL=0
MOVL C00876 V=800.0 PL=0
MOVL C00877 V=800.0 PL=0
MOVL C00878 V=800.0 PL=0
MOVL C00879 V=800.0 PL=0
MOVL C00880 V=800.0 PL=0
MOVL C00881 V=800.0 PL=0
MOVL C00882 V=800.0 PL=0
MOVL C00883 V=800.0 PL=0
MOVL C00884 V=800.0 PL=0
MOVL C00885 V=800.0 PL=0
MOVL C00886 V=800.0 PL=0
MOVL C00887 V=800.0 PL=0
MOVL C00888 V=800.0 PL=0
MOVL C00889 V=800.0 PL=0
MOVL C00890 V=800.0 PL=0
MOVL C00891 V=800.0 PL=0
MOVL C00892 V=800.0 PL=0
MOVL C00893 V=800.0 PL=0
MOVL C00894 V=800.0 PL=0
MOVL C00895 V=800.0 PL=0
MOVL C00896 V=800.0 PL=0
MOVL C00897 V=800.0 PL=0
MOVL C00898 V=800.0 PL=0
MOVL C00899 V=800.0 PL=0
MOVL C00900 V=800.0 PL=0
MOVL C00901 V=800.0 PL=0
MOVL C00902 V=800.0 PL=0
MOVL C00903 V=800.0 PL=0
MOVL C00904 V=800.0 PL=0
MOVL C00905 V=800.0 PL=0
MOVL C00906 V=800.0 PL=0
MOVL C00907 V=800.0 PL=0
MOVL C00908 V=800.0 PL=0
MOVL C00909 V=800.0 PL=0
MOVL C00910 V=800.0 PL=0
MOVL C00911 V=800.0 PL=0
MOVL C00912 V=800.0 PL=0
MOVL C00913 V=800.0 PL=0
MOVL C00914 V=800.0 PL=0
MOVL C00915 V=800.0 PL=0
MOVL C00916 V=800.0 PL=0
MOVL C00917 V=800.0 PL=0
MOVL C00918 V=800.0 PL=0
MOVL C00919 V=800.0 PL=0
MOVL C00920 V=800.0 PL=0
MOVL C00921 V=800.0 PL=0
MOVL C00922 V=800.0 PL=0
MOVL C00923 V=800.0 PL=0
MOVL C00924 V=800.0 PL=0
MOVL C00925 V=800.0 PL=0
MOVL C00926 V=800.0 PL=0
MOVL C00927 V=800.0 PL=0
MOVL C00928 V=800.0 PL=0
MOVL C00929 V=800.0 PL=0
MOVL C00930 V=800.0 PL=0
MOVL C00931 V=800.0 PL=0
MOVL C00932 V=800.0 PL=0
MOVL C00933 V=800.0 PL=0
MOVL C00934 V=800.0 PL=0
MOVL C00935 V=800.0 PL=0
MOVL C00936 V=800.0 PL=0
MOVL C00937 V=800.0 PL=0
MOVL C00938 V=800.0 PL=0
MOVL C00939 V=800.0 PL=0
MOVL C00940 V=800.0 PL=0
MOVL C00941 V=800.0 PL=0
MOVL C00942 V=800.0 PL=0
MOVL C00943 V=800.0 PL=0
MOVL C00944 V=800.0 PL=0
MOVL C00945 V=800.0 PL=0
MOVL C00946 V=800.0 PL=0
MOVL C00947 V=800.0 PL=0
MOVL C00948 V=800.0 PL=0
MOVL C00949 V=800.0 PL=0
MOVL C00950 V=800.0 PL=0
MOVL C00951 V=800.0 PL=0
MOVL C00952 V=800.0 PL=0
MOVL C00953 V=800.0 PL=0
MOVL C00954 V=800.0 PL=0
MOVL C00955 V=800.0 PL=0
MOVL C00956 V=800.0 PL=0
MOVL C00957 V=800.0 PL=0
MOVL C00958 V=800.0 PL=0
MOVL C00959 V=800.0 PL=0
MOVL C00960 V=800.0 PL=0
MOVL C00961 V=800.0 PL=0
MOVL C00962 V=800.0 PL=0
MOVL C00963 V=800.0 PL=0
MOVL C00964 V=800.0 PL=0
MOVL C00965 V=800.0 PL=0
MOVL C00966 V=800.0 PL=0
MOVL C00967 V=800.0 PL=0
MOVL C00968 V=800.0 PL=0
MOVL C00969 V=800.0 PL=0
MOVL C00970 V=800.0 PL=0
MOVL C00971 V=800.0 PL=0
MOVL C00972 V=800.0 PL=0
MOVL C00973 V=800.0 PL=0
MOVL C00974 V=800.0 PL=0
MOVL C00975 V=800.0 PL=0
MOVL C00976 V=800.0 PL=0
MOVL C00977 V=800.0 PL=0
MOVL C00978 V=800.0 PL=0
MOVL C00979 V=800.0 PL=0
MOVL C00980 V=800.0 PL=0
MOVL C00981 V=800.0 PL=0
MOVL C00982 V=800.0 PL=0
MOVL C00983 V=800.0 PL=0
MOVL C00984 V=800.0 PL=0
MOVL C00985 V=800.0 PL=0
MOVL C00986 V=800.0 PL=0
MOVL C00987 V=800.0 PL=0
MOVL C00988 V=800.0 PL=0
MOVL C00989 V=800.0 PL=0
MOVL C00990 V=800.0 PL=0
MOVL C00991 V=800.0 PL=0
MOVL C00992 V=800.0 PL=0
MOVL C00993 V=800.0 PL=0
MOVL C00994 V=800.0 PL=0
MOVL C00995 V=800.0 PL=0
MOVL C00996 V=800.0 PL=0
MOVL C00997 V=800.0 PL=0
MOVL C00998 V=800.0 PL=0
MOVL C00999 V=800.0 PL=0
MOVL C01000 V=800.0 PL=0
MOVL C01001 V=800.0 PL=0
MOVL C01002 V=800.0 PL=0
MOVL C01003 V=800.0 PL=0
MOVL C01004 V=800.0 PL=0
MOVL C01005 V=800.0 PL=0
MOVL C01006 V=800.0 PL=0
MOVL C01007 V=800.0 PL=0
MOVL C01008 V=800.0 PL=0
MOVL C01009 V=800.0 PL=0
MOVL C01010 V=800.0 PL=0
MOVL C01011 V=800.0 PL=0
MOVL C01012 V=800.0 PL=0
MOVL C01013 V=800.0 PL=0
MOVL C01014 V=800.0 PL=0
MOVL C01015 V=800.0 PL=0
MOVL C01016 V=800.0 PL=0
MOVL C01017 V=800.0 PL=0
MOVL C01018 V=800.0 PL=0
MOVL C01019 V=800.0 PL=0
MOVL C01020 V=800.0 PL=0
MOVL C01021 V=800.0 PL=0
MOVL C01022 V=800.0 PL=0
MOVL C01023 V=800.0 PL=0
MOVL C01024 V=800.0 PL=0
MOVL C01025 V=800.0 PL=0
MOVL C01026 V=800.0 PL=0
MOVL C01027 V=800.0 PL=0
MOVL C01028 V=800.0 PL=0
MOVL C01029 V=800.0 PL=0
MOVL C01030 V=800.0 PL=0
MOVL C01031 V=800.0 PL=0
MOVL C01032 V=800.0 PL=0
MOVL C01033 V=800.0 PL=0
MOVL C01034 V=800.0 PL=0
MOVL C01035 V=800.0 PL=0
MOVL C01036 V=800.0 PL=0
MOVL C01037 V=800.0 PL=0
MOVL C01038 V=800.0 PL=0
MOVL C01039 V=800.0 PL=0
MOVL C01040 V=800.0 PL=0
MOVL C01041 V=800.0 PL=0
MOVL C01042 V=800.0 PL=0
MOVL C01043 V=800.0 PL=0
MOVL C01044 V=800.0 PL=0
MOVL C01045 V=800.0 PL=0
MOVL C01046 V=800.0 PL=0
MOVL C01047 V=800.0 PL=0
MOVL C01048 V=800.0 PL=0
MOVL C01049 V=800.0 PL=0
MOVL C01050 V=800.0 PL=0
MOVL C01051 V=800.0 PL=0
MOVL C01052 V=800.0 PL=0
MOVL C01053 V=800.0 PL=0
MOVL C01054 V=800.0 PL=0
MOVL C01055 V=800.0 PL=0
MOVL C01056 V=800.0 PL=0
MOVL C01057 V=800.0 PL=0
MOVL C01058 V=800.0 PL=0
MOVL C01059 V=800.0 PL=0
MOVL C01060 V=800.0 PL=0
MOVL C01061 V=800.0 PL=0
MOVL C01062 V=800.0 PL=0
MOVL C01063 V=800.0 PL=0
MOVL C01064 V=800.0 PL=0
MOVL C01065 V=800.0 PL=0
MOVL C01066 V=800.0 PL=0
MOVL C01067 V=800.0 PL=0
MOVL C01068 V=800.0 PL=0
MOVL C01069 V=800.0 PL=0
MOVL C01070 V=800.0 PL=0
MOVL C01071 V=800.0 PL=0
MOVL C01072 V=800.0 PL=0
MOVL C01073 V=800.0 PL=0
MOVL C01074 V=800.0 PL=0
MOVL C01075 V=800.0 PL=0
MOVL C01076 V=800.0 PL=0
MOVL C01077 V=800.0 PL=0
MOVL C01078 V=800.0 PL=0
MOVL C01079 V=800.0 PL=0
MOVL C01080 V=800.0 PL=0
MOVL C01081 V=800.0 PL=0
MOVL C01082 V=800.0 PL=0
MOVL C01083 V=800.0 PL=0
MOVL C01084 V=800.0 PL=0
MOVL C01085 V=800.0 PL=0
MOVL C01086 V=800.0 PL=0
MOVL C01087 V=800.0 PL=0
MOVL C01088 V=800.0 PL=0
MOVL C01089 V=800.0 PL=0
MOVL C01090 V=800.0 PL=0
MOVL C01091 V=800.0 PL=0
MOVL C01092 V=800.0 PL=0
MOVL C01093 V=800.0 PL=0
MOVL C01094 V=800.0 PL=0
MOVL C01095 V=800.0 PL=0
MOVL C01096 V=800.0 PL=0
MOVL C01097 V=800.0 PL=0
MOVL C01098 V=800.0 PL=0
MOVL C01099 V=800.0 PL=0
MOVL C01100 V=800.0 PL=0
MOVL C01101 V=800.0 PL=0
MOVL C01102 V=800.0 PL=0
MOVL C01103 V=800.0 PL=0
MOVL C01104 V=800.0 PL=0
MOVL C01105 V=800.0 PL=0
MOVL C01106 V=800.0 PL=0
MOVL C01107 V=800.0 PL=0
MOVL C01108 V=800.0 PL=0
MOVL C01109 V=800.0 PL=0
MOVL C01110 V=800.0 PL=0
MOVL C01111 V=800.0 PL=0
MOVL C01112 V=800.0 PL=0
MOVL C01113 V=800.0 PL=0
MOVL C01114 V=800.0 PL=0
MOVL C01115 V=800.0 PL=0
MOVL C01116 V=800.0 PL=0
MOVL C01117 V=800.0 PL=0
MOVL C01118 V=800.0 PL=0
MOVL C01119 V=800.0 PL=0
MOVL C01120 V=800.0 PL=0
MOVL C01121 V=800.0 PL=0
MOVL C01122 V=800.0 PL=0
MOVL C01123 V=800.0 PL=0
MOVL C01124 V=800.0 PL=0
MOVL C01125 V=800.0 PL=0
MOVL C01126 V=800.0 PL=0
MOVL C01127 V=800.0 PL=0
MOVL C01128 V=800.0 PL=0
MOVL C01129 V=800.0 PL=0
MOVL C01130 V=800.0 PL=0
MOVL C01131 V=800.0 PL=0
MOVL C01132 V=800.0 PL=0
MOVL C01133 V=800.0 PL=0
MOVL C01134 V=800.0 PL=0
MOVL C01135 V=800.0 PL=0
MOVL C01136 V=800.0 PL=0
MOVL C01137 V=800.0 PL=0
MOVL C01138 V=800.0 PL=0
MOVL C01139 V=800.0 PL=0
MOVL C01140 V=800.0 PL=0
MOVL C01141 V=800.0 PL=0
MOVL C01142 V=800.0 PL=0
MOVL C01143 V=800.0 PL=0
MOVL C01144 V=800.0 PL=0
MOVL C01145 V=800.0 PL=0
MOVL C01146 V=800.0 PL=0
MOVL C01147 V=800.0 PL=0
MOVL C01148 V=800.0 PL=0
MOVL C01149 V=800.0 PL=0
MOVL C01150 V=800.0 PL=0
MOVL C01151 V=800.0 PL=0
MOVL C01152 V=800.0 PL=0
MOVL C01153 V=800.0 PL=0
MOVL C01154 V=800.0 PL=0
MOVL C01155 V=800.0 PL=0
MOVL C01156 V=800.0 PL=0
MOVL C01157 V=800.0 PL=0
MOVL C01158 V=800.0 PL=0
MOVL C01159 V=800.0 PL=0
MOVL C01160 V=800.0 PL=0
MOVL C01161 V=800.0 PL=0
MOVL C01162 V=800.0 PL=0
MOVL C01163 V=800.0 PL=0
MOVL C01164 V=800.0 PL=0
MOVL C01165 V=800.0 PL=0
MOVL C01166 V=800.0 PL=0
MOVL C01167 V=800.0 PL=0
MOVL C01168 V=800.0 PL=0
MOVL C01169 V=800.0 PL=0
MOVL C01170 V=800.0 PL=0
MOVL C01171 V=800.0 PL=0
MOVL C01172 V=800.0 PL=0
MOVL C01173 V=800.0 PL=0
MOVL C01174 V=800.0 PL=0
MOVL C01175 V=800.0 PL=0
MOVL C01176 V=800.0 PL=0
MOVL C01177 V=800.0 PL=0
MOVL C01178 V=800.0 PL=0
MOVL C01179 V=800.0 PL=0
MOVL C01180 V=800.0 PL=0
MOVL C01181 V=800.0 PL=0
MOVL C01182 V=800.0 PL=0
MOVL C01183 V=800.0 PL=0
MOVL C01184 V=800.0 PL=0
MOVL C01185 V=800.0 PL=0
MOVL C01186 V=800.0 PL=0
MOVL C01187 V=800.0 PL=0
MOVL C01188 V=800.0 PL=0
MOVL C01189 V=800.0 PL=0
MOVL C01190 V=800.0 PL=0
MOVL C01191 V=800.0 PL=0
MOVL C01192 V=800.0 PL=0
MOVL C01193 V=800.0 PL=0
MOVL C01194 V=800.0 PL=0
MOVL C01195 V=800.0 PL=0
MOVL C01196 V=800.0 PL=0
MOVL C01197 V=800.0 PL=0
MOVL C01198 V=800.0 PL=0
MOVL C01199 V=800.0 PL=0
MOVL C01200 V=800.0 PL=0
MOVL C01201 V=800.0 PL=0
MOVL C01202 V=800.0 PL=0
MOVL C01203 V=800.0 PL=0
MOVL C01204 V=800.0 PL=0
MOVL C01205 V=800.0 PL=0
MOVL C01206 V=800.0 PL=0
MOVL C01207 V=800.0 PL=0
MOVL C01208 V=800.0 PL=0
MOVL C01209 V=800.0 PL=0
MOVL C01210 V=800.0 PL=0
MOVL C01211 V=800.0 PL=0
MOVL C01212 V=800.0 PL=0
MOVL C01213 V=800.0 PL=0
MOVL C01214 V=800.0 PL=0
MOVL C01215 V=800.0 PL=0
MOVL C01216 V=800.0 PL=0
MOVL C01217 V=800.0 PL=0
MOVL C01218 V=800.0 PL=0
MOVL C01219 V=800.0 PL=0
MOVL C01220 V=800.0 PL=0
MOVL C01221 V=800.0 PL=0
MOVL C01222 V=800.0 PL=0
MOVL C01223 V=800.0 PL=0
MOVL C01224 V=800.0 PL=0
MOVL C01225 V=800.0 PL=0
MOVL C01226 V=800.0 PL=0
MOVL C01227 V=800.0 PL=0
MOVL C01228 V=800.0 PL=0
MOVL C01229 V=800.0 PL=0
MOVL C01230 V=800.0 PL=0
MOVL C01231 V=800.0 PL=0
MOVL C01232 V=800.0 PL=0
MOVL C01233 V=800.0 PL=0
MOVL C01234 V=800.0 PL=0
MOVL C01235 V=800.0 PL=0
MOVL C01236 V=800.0 PL=0
MOVL C01237 V=800.0 PL=0
MOVL C01238 V=800.0 PL=0
MOVL C01239 V=800.0 PL=0
MOVL C01240 V=800.0 PL=0
MOVL C01241 V=800.0 PL=0
MOVL C01242 V=800.0 PL=0
MOVL C01243 V=800.0 PL=0
MOVL C01244 V=800.0 PL=0
MOVL C01245 V=800.0 PL=0
MOVL C01246 V=800.0 PL=0
MOVL C01247 V=800.0 PL=0
MOVL C01248 V=800.0 PL=0
MOVL C01249 V=800.0 PL=0
MOVL C01250 V=800.0 PL=0
MOVL C01251 V=800.0 PL=0
MOVL C01252 V=800.0 PL=0
MOVL C01253 V=800.0 PL=0
MOVL C01254 V=800.0 PL=0
MOVL C01255 V=800.0 PL=0
MOVL C01256 V=800.0 PL=0
MOVL C01257 V=800.0 PL=0
MOVL C01258 V=800.0 PL=0
MOVL C01259 V=800.0 PL=0
MOVL C01260 V=800.0 PL=0
MOVL C01261 V=800.0 PL=0
MOVL C01262 V=800.0 PL=0
MOVL C01263 V=800.0 PL=0
MOVL C01264 V=800.0 PL=0
MOVL C01265 V=800.0 PL=0
MOVL C01266 V=800.0 PL=0
MOVL C01267 V=800.0 PL=0
MOVL C01268 V=800.0 PL=0
MOVL C01269 V=800.0 PL=0
MOVL C01270 V=800.0 PL=0
MOVL C01271 V=800.0 PL=0
MOVL C01272 V=800.0 PL=0
MOVL C01273 V=800.0 PL=0
MOVL C01274 V=800.0 PL=0
MOVL C01275 V=800.0 PL=0
MOVL C01276 V=800.0 PL=0
MOVL C01277 V=800.0 PL=0
MOVL C01278 V=800.0 PL=0
MOVL C01279 V=800.0 PL=0
MOVL C01280 V=800.0 PL=0
MOVL C01281 V=800.0 PL=0
MOVL C01282 V=800.0 PL=0
MOVL C01283 V=800.0 PL=0
MOVL C01284 V=800.0 PL=0
MOVL C01285 V=800.0 PL=0
MOVL C01286 V=800.0 PL=0
MOVL C01287 V=800.0 PL=0
MOVL C01288 V=800.0 PL=0
MOVL C01289 V=800.0 PL=0
MOVL C01290 V=800.0 PL=0
MOVL C01291 V=800.0 PL=0
MOVL C01292 V=800.0 PL=0
MOVL C01293 V=800.0 PL=0
MOVL C01294 V=800.0 PL=0
MOVL C01295 V=800.0 PL=0
MOVL C01296 V=800.0 PL=0
MOVL C01297 V=800.0 PL=0
MOVL C01298 V=800.0 PL=0
MOVL C01299 V=800.0 PL=0
MOVL C01300 V=800.0 PL=0
MOVL C01301 V=800.0 PL=0
MOVL C01302 V=800.0 PL=0
MOVL C01303 V=800.0 PL=0
MOVL C01304 V=800.0 PL=0
MOVL C01305 V=800.0 PL=0
MOVL C01306 V=800.0 PL=0
MOVL C01307 V=800.0 PL=0
MOVL C01308 V=800.0 PL=0
MOVL C01309 V=800.0 PL=0
MOVL C01310 V=800.0 PL=0
MOVL C01311 V=800.0 PL=0
MOVL C01312 V=800.0 PL=0
MOVL C01313 V=800.0 PL=0
MOVL C01314 V=800.0 PL=0
MOVL C01315 V=800.0 PL=0
MOVL C01316 V=800.0 PL=0
MOVL C01317 V=800.0 PL=0
MOVL C01318 V=800.0 PL=0
MOVL C01319 V=800.0 PL=0
MOVL C01320 V=800.0 PL=0
MOVL C01321 V=800.0 PL=0
MOVL C01322 V=800.0 PL=0
MOVL C01323 V=800.0 PL=0
MOVL C01324 V=800.0 PL=0
MOVL C01325 V=800.0 PL=0
MOVL C01326 V=800.0 PL=0
MOVL C01327 V=800.0 PL=0
MOVL C01328 V=800.0 PL=0
MOVL C01329 V=800.0 PL=0
MOVL C01330 V=800.0 PL=0
MOVL C01331 V=800.0 PL=0
MOVL C01332 V=800.0 PL=0
MOVL C01333 V=800.0 PL=0
MOVL C01334 V=800.0 PL=0
MOVL C01335 V=800.0 PL=0
MOVL C01336 V=800.0 PL=0
MOVL C01337 V=800.0 PL=0
MOVL C01338 V=800.0 PL=0
MOVL C01339 V=800.0 PL=0
MOVL C01340 V=800.0 PL=0
MOVL C01341 V=800.0 PL=0
MOVL C01342 V=800.0 PL=0
MOVL C01343 V=800.0 PL=0
MOVL C01344 V=800.0 PL=0
MOVL C01345 V=800.0 PL=0
MOVL C01346 V=800.0 PL=0
MOVL C01347 V=800.0 PL=0
MOVL C01348 V=800.0 PL=0
MOVL C01349 V=800.0 PL=0
MOVL C01350 V=800.0 PL=0
MOVL C01351 V=800.0 PL=0
MOVL C01352 V=800.0 PL=0
MOVL C01353 V=800.0 PL=0
MOVL C01354 V=800.0 PL=0
MOVL C01355 V=800.0 PL=0
MOVL C01356 V=800.0 PL=0
MOVL C01357 V=800.0 PL=0
MOVL C01358 V=800.0 PL=0
MOVL C01359 V=800.0 PL=0
MOVL C01360 V=800.0 PL=0
MOVL C01361 V=800.0 PL=0
MOVL C01362 V=800.0 PL=0
MOVL C01363 V=800.0 PL=0
MOVL C01364 V=800.0 PL=0
MOVL C01365 V=800.0 PL=0
MOVL C01366 V=800.0 PL=0
MOVL C01367 V=800.0 PL=0
MOVL C01368 V=800.0 PL=0
MOVL C01369 V=800.0 PL=0
MOVL C01370 V=800.0 PL=0
MOVL C01371 V=800.0 PL=0
MOVL C01372 V=800.0 PL=0
MOVL C01373 V=800.0 PL=0
MOVL C01374 V=800.0 PL=0
MOVL C01375 V=800.0 PL=0
MOVL C01376 V=800.0 PL=0
MOVL C01377 V=800.0 PL=0
MOVL C01378 V=800.0 PL=0
MOVL C01379 V=800.0 PL=0
MOVL C01380 V=800.0 PL=0
MOVL C01381 V=800.0 PL=0
MOVL C01382 V=800.0 PL=0
MOVL C01383 V=800.0 PL=0
MOVL C01384 V=800.0 PL=0
MOVL C01385 V=800.0 PL=0
MOVL C01386 V=800.0 PL=0
MOVL C01387 V=800.0 PL=0
MOVL C01388 V=800.0 PL=0
MOVL C01389 V=800.0 PL=0
MOVL C01390 V=800.0 PL=0
MOVL C01391 V=800.0 PL=0
MOVL C01392 V=800.0 PL=0
MOVL C01393 V=800.0 PL=0
MOVL C01394 V=800.0 PL=0
MOVL C01395 V=800.0 PL=0
MOVL C01396 V=800.0 PL=0
MOVL C01397 V=800.0 PL=0
MOVL C01398 V=800.0 PL=0
MOVL C01399 V=800.0 PL=0
MOVL C01400 V=800.0 PL=0
MOVL C01401 V=800.0 PL=0
MOVL C01402 V=800.0 PL=0
MOVL C01403 V=800.0 PL=0
MOVL C01404 V=800.0 PL=0
MOVL C01405 V=800.0 PL=0
MOVL C01406 V=800.0 PL=0
MOVL C01407 V=800.0 PL=0
MOVL C01408 V=800.0 PL=0
MOVL C01409 V=800.0 PL=0
MOVL C01410 V=800.0 PL=0
MOVL C01411 V=800.0 PL=0
MOVL C01412 V=800.0 PL=0
MOVL C01413 V=800.0 PL=0
MOVL C01414 V=800.0 PL=0
MOVL C01415 V=800.0 PL=0
MOVL C01416 V=800.0 PL=0
MOVL C01417 V=800.0 PL=0
MOVL C01418 V=800.0 PL=0
MOVL C01419 V=800.0 PL=0
MOVL C01420 V=800.0 PL=0
MOVL C01421 V=800.0 PL=0
MOVL C01422 V=800.0 PL=0
MOVL C01423 V=800.0 PL=0
MOVL C01424 V=800.0 PL=0
MOVL C01425 V=800.0 PL=0
MOVL C01426 V=800.0 PL=0
MOVL C01427 V=800.0 PL=0
MOVL C01428 V=800.0 PL=0
MOVL C01429 V=800.0 PL=0
MOVL C01430 V=800.0 PL=0
MOVL C01431 V=800.0 PL=0
MOVL C01432 V=800.0 PL=0
MOVL C01433 V=800.0 PL=0
MOVL C01434 V=800.0 PL=0
MOVL C01435 V=800.0 PL=0
MOVL C01436 V=800.0 PL=0
MOVL C01437 V=800.0 PL=0
MOVL C01438 V=800.0 PL=0
MOVL C01439 V=800.0 PL=0
MOVL C01440 V=800.0 PL=0
MOVL C01441 V=800.0 PL=0
MOVL C01442 V=800.0 PL=0
MOVL C01443 V=800.0 PL=0
MOVL C01444 V=800.0 PL=0
MOVL C01445 V=800.0 PL=0
MOVL C01446 V=800.0 PL=0
MOVL C01447 V=800.0 PL=0
MOVL C01448 V=800.0 PL=0
MOVL C01449 V=800.0 PL=0
MOVL C01450 V=800.0 PL=0
MOVL C01451 V=800.0 PL=0
MOVL C01452 V=800.0 PL=0
MOVL C01453 V=800.0 PL=0
MOVL C01454 V=800.0 PL=0
MOVL C01455 V=800.0 PL=0
MOVL C01456 V=800.0 PL=0
MOVL C01457 V=800.0 PL=0
MOVL C01458 V=800.0 PL=0
MOVL C01459 V=800.0 PL=0
MOVL C01460 V=800.0 PL=0
MOVL C01461 V=800.0 PL=0
MOVL C01462 V=800.0 PL=0
MOVL C01463 V=800.0 PL=0
MOVL C01464 V=800.0 PL=0
MOVL C01465 V=800.0 PL=0
MOVL C01466 V=800.0 PL=0
MOVL C01467 V=800.0 PL=0
MOVL C01468 V=800.0 PL=0
MOVL C01469 V=800.0 PL=0
MOVL C01470 V=800.0 PL=0
MOVL C01471 V=800.0 PL=0
MOVL C01472 V=800.0 PL=0
MOVL C01473 V=800.0 PL=0
MOVL C01474 V=800.0 PL=0
MOVL C01475 V=800.0 PL=0
MOVL C01476 V=800.0 PL=0
MOVL C01477 V=800.0 PL=0
MOVL C01478 V=800.0 PL=0
MOVL C01479 V=800.0 PL=0
MOVL C01480 V=800.0 PL=0
MOVL C01481 V=800.0 PL=0
MOVL C01482 V=800.0 PL=0
MOVL C01483 V=800.0 PL=0
MOVL C01484 V=800.0 PL=0
MOVL C01485 V=800.0 PL=0
MOVL C01486 V=800.0 PL=0
MOVL C01487 V=800.0 PL=0
MOVL C01488 V=800.0 PL=0
MOVL C01489 V=800.0 PL=0
MOVL C01490 V=800.0 PL=0
MOVL C01491 V=800.0 PL=0
MOVL C01492 V=800.0 PL=0
MOVL C01493 V=800.0 PL=0
MOVL C01494 V=800.0 PL=0
MOVL C01495 V=800.0 PL=0
MOVL C01496 V=800.0 PL=0
MOVL C01497 V=800.0 PL=0
MOVL C01498 V=800.0 PL=0
MOVL C01499 V=800.0 PL=0
MOVL C01500 V=800.0 PL=0
MOVL C01501 V=800.0 PL=0
MOVL C01502 V=800.0 PL=0
MOVL C01503 V=800.0 PL=0
MOVL C01504 V=800.0 PL=0
MOVL C01505 V=800.0 PL=0
MOVL C01506 V=800.0 PL=0
MOVL C01507 V=800.0 PL=0
MOVL C01508 V=800.0 PL=0
MOVL C01509 V=800.0 PL=0
MOVL C01510 V=800.0 PL=0
MOVL C01511 V=800.0 PL=0
MOVL C01512 V=800.0 PL=0
MOVL C01513 V=800.0 PL=0
MOVL C01514 V=800.0 PL=0
MOVL C01515 V=800.0 PL=0
MOVL C01516 V=800.0 PL=0
MOVL C01517 V=800.0 PL=0
MOVL C01518 V=800.0 PL=0
MOVL C01519 V=800.0 PL=0
MOVL C01520 V=800.0 PL=0
MOVL C01521 V=800.0 PL=0
MOVL C01522 V=800.0 PL=0
MOVL C01523 V=800.0 PL=0
MOVL C01524 V=800.0 PL=0
MOVL C01525 V=800.0 PL=0
MOVL C01526 V=800.0 PL=0
MOVL C01527 V=800.0 PL=0
MOVL C01528 V=800.0 PL=0
MOVL C01529 V=800.0 PL=0
MOVL C01530 V=800.0 PL=0
MOVL C01531 V=800.0 PL=0
MOVL C01532 V=800.0 PL=0
MOVL C01533 V=800.0 PL=0
MOVL C01534 V=800.0 PL=0
MOVL C01535 V=800.0 PL=0
MOVL C01536 V=800.0 PL=0
MOVL C01537 V=800.0 PL=0
MOVL C01538 V=800.0 PL=0
MOVL C01539 V=800.0 PL=0
MOVL C01540 V=800.0 PL=0
MOVL C01541 V=800.0 PL=0
MOVL C01542 V=800.0 PL=0
MOVL C01543 V=800.0 PL=0
MOVL C01544 V=800.0 PL=0
MOVL C01545 V=800.0 PL=0
MOVL C01546 V=800.0 PL=0
MOVL C01547 V=800.0 PL=0
MOVL C01548 V=800.0 PL=0
MOVL C01549 V=800.0 PL=0
MOVL C01550 V=800.0 PL=0
MOVL C01551 V=800.0 PL=0
MOVL C01552 V=800.0 PL=0
MOVL C01553 V=800.0 PL=0
MOVL C01554 V=800.0 PL=0
MOVL C01555 V=800.0 PL=0
MOVL C01556 V=800.0 PL=0
MOVL C01557 V=800.0 PL=0
MOVL C01558 V=800.0 PL=0
MOVL C01559 V=800.0 PL=0
MOVL C01560 V=800.0 PL=0
MOVL C01561 V=800.0 PL=0
MOVL C01562 V=800.0 PL=0
MOVL C01563 V=800.0 PL=0
MOVL C01564 V=800.0 PL=0
MOVL C01565 V=800.0 PL=0
MOVL C01566 V=800.0 PL=0
MOVL C01567 V=800.0 PL=0
MOVL C01568 V=800.0 PL=0
MOVL C01569 V=800.0 PL=0
MOVL C01570 V=800.0 PL=0
MOVL C01571 V=800.0 PL=0
MOVL C01572 V=800.0 PL=0
MOVL C01573 V=800.0 PL=0
MOVL C01574 V=800.0 PL=0
MOVL C01575 V=800.0 PL=0
MOVL C01576 V=800.0 PL=0
MOVL C01577 V=800.0 PL=0
MOVL C01578 V=800.0 PL=0
MOVL C01579 V=800.0 PL=0
MOVL C01580 V=800.0 PL=0
MOVL C01581 V=800.0 PL=0
MOVL C01582 V=800.0 PL=0
MOVL C01583 V=800.0 PL=0
MOVL C01584 V=800.0 PL=0
MOVL C01585 V=800.0 PL=0
MOVL C01586 V=800.0 PL=0
MOVL C01587 V=800.0 PL=0
MOVL C01588 V=800.0 PL=0
MOVL C01589 V=800.0 PL=0
MOVL C01590 V=800.0 PL=0
MOVL C01591 V=800.0 PL=0
MOVL C01592 V=800.0 PL=0
MOVL C01593 V=800.0 PL=0
MOVL C01594 V=800.0 PL=0
MOVL C01595 V=800.0 PL=0
MOVL C01596 V=800.0 PL=0
MOVL C01597 V=800.0 PL=0
MOVL C01598 V=800.0 PL=0
MOVL C01599 V=800.0 PL=0
MOVL C01600 V=800.0 PL=0
MOVL C01601 V=800.0 PL=0
MOVL C01602 V=800.0 PL=0
MOVL C01603 V=800.0 PL=0
MOVL C01604 V=800.0 PL=0
MOVL C01605 V=800.0 PL=0
MOVL C01606 V=800.0 PL=0
MOVL C01607 V=800.0 PL=0
MOVL C01608 V=800.0 PL=0
MOVL C01609 V=800.0 PL=0
MOVL C01610 V=800.0 PL=0
MOVL C01611 V=800.0 PL=0
MOVL C01612 V=800.0 PL=0
MOVL C01613 V=800.0 PL=0
MOVL C01614 V=800.0 PL=0
MOVL C01615 V=800.0 PL=0
MOVL C01616 V=800.0 PL=0
MOVL C01617 V=800.0 PL=0
MOVL C01618 V=800.0 PL=0
MOVL C01619 V=800.0 PL=0
MOVL C01620 V=800.0 PL=0
MOVL C01621 V=800.0 PL=0
MOVL C01622 V=800.0 PL=0
MOVL C01623 V=800.0 PL=0
MOVL C01624 V=800.0 PL=0
MOVL C01625 V=800.0 PL=0
MOVL C01626 V=800.0 PL=0
MOVL C01627 V=800.0 PL=0
MOVL C01628 V=800.0 PL=0
MOVL C01629 V=800.0 PL=0
MOVL C01630 V=800.0 PL=0
MOVL C01631 V=800.0 PL=0
MOVL C01632 V=800.0 PL=0
MOVL C01633 V=800.0 PL=0
MOVL C01634 V=800.0 PL=0
MOVL C01635 V=800.0 PL=0
MOVL C01636 V=800.0 PL=0
MOVL C01637 V=800.0 PL=0
MOVL C01638 V=800.0 PL=0
MOVL C01639 V=800.0 PL=0
MOVL C01640 V=800.0 PL=0
MOVL C01641 V=800.0 PL=0
MOVL C01642 V=800.0 PL=0
MOVL C01643 V=800.0 PL=0
MOVL C01644 V=800.0 PL=0
MOVL C01645 V=800.0 PL=0
MOVL C01646 V=800.0 PL=0
MOVL C01647 V=800.0 PL=0
MOVL C01648 V=800.0 PL=0
MOVL C01649 V=800.0 PL=0
MOVL C01650 V=800.0 PL=0
MOVL C01651 V=800.0 PL=0
MOVL C01652 V=800.0 PL=0
MOVL C01653 V=800.0 PL=0
MOVL C01654 V=800.0 PL=0
MOVL C01655 V=800.0 PL=0
MOVL C01656 V=800.0 PL=0
MOVL C01657 V=800.0 PL=0
MOVL C01658 V=800.0 PL=0
MOVL C01659 V=800.0 PL=0
MOVL C01660 V=800.0 PL=0
MOVL C01661 V=800.0 PL=0
MOVL C01662 V=800.0 PL=0
MOVL C01663 V=800.0 PL=0
MOVL C01664 V=800.0 PL=0
MOVL C01665 V=800.0 PL=0
MOVL C01666 V=800.0 PL=0
MOVL C01667 V=800.0 PL=0
MOVL C01668 V=800.0 PL=0
MOVL C01669 V=800.0 PL=0
MOVL C01670 V=800.0 PL=0
MOVL C01671 V=800.0 PL=0
MOVL C01672 V=800.0 PL=0
MOVL C01673 V=800.0 PL=0
MOVL C01674 V=800.0 PL=0
MOVL C01675 V=800.0 PL=0
MOVL C01676 V=800.0 PL=0
MOVL C01677 V=800.0 PL=0
MOVL C01678 V=800.0 PL=0
MOVL C01679 V=800.0 PL=0
MOVL C01680 V=800.0 PL=0
MOVL C01681 V=800.0 PL=0
MOVL C01682 V=800.0 PL=0
MOVL C01683 V=800.0 PL=0
MOVL C01684 V=800.0 PL=0
MOVL C01685 V=800.0 PL=0
MOVL C01686 V=800.0 PL=0
MOVL C01687 V=800.0 PL=0
MOVL C01688 V=800.0 PL=0
MOVL C01689 V=800.0 PL=0
MOVL C01690 V=800.0 PL=0
MOVL C01691 V=800.0 PL=0
MOVL C01692 V=800.0 PL=0
MOVL C01693 V=800.0 PL=0
MOVL C01694 V=800.0 PL=0
MOVL C01695 V=800.0 PL=0
MOVL C01696 V=800.0 PL=0
MOVL C01697 V=800.0 PL=0
MOVL C01698 V=800.0 PL=0
MOVL C01699 V=800.0 PL=0
MOVL C01700 V=800.0 PL=0
MOVL C01701 V=800.0 PL=0
MOVL C01702 V=800.0 PL=0
MOVL C01703 V=800.0 PL=0
MOVL C01704 V=800.0 PL=0
MOVL C01705 V=800.0 PL=0
MOVL C01706 V=800.0 PL=0
MOVL C01707 V=800.0 PL=0
MOVL C01708 V=800.0 PL=0
MOVL C01709 V=800.0 PL=0
MOVL C01710 V=800.0 PL=0
MOVL C01711 V=800.0 PL=0
MOVL C01712 V=800.0 PL=0
MOVL C01713 V=800.0 PL=0
MOVL C01714 V=800.0 PL=0
MOVL C01715 V=800.0 PL=0
MOVL C01716 V=800.0 PL=0
MOVL C01717 V=800.0 PL=0
MOVL C01718 V=800.0 PL=0
MOVL C01719 V=800.0 PL=0
MOVL C01720 V=800.0 PL=0
MOVL C01721 V=800.0 PL=0
MOVL C01722 V=800.0 PL=0
MOVL C01723 V=800.0 PL=0
MOVL C01724 V=800.0 PL=0
MOVL C01725 V=800.0 PL=0
MOVL C01726 V=800.0 PL=0
MOVL C01727 V=800.0 PL=0
MOVL C01728 V=800.0 PL=0
MOVL C01729 V=800.0 PL=0
MOVL C01730 V=800.0 PL=0
MOVL C01731 V=800.0 PL=0
MOVL C01732 V=800.0 PL=0
MOVL C01733 V=800.0 PL=0
MOVL C01734 V=800.0 PL=0
MOVL C01735 V=800.0 PL=0
MOVL C01736 V=800.0 PL=0
MOVL C01737 V=800.0 PL=0
MOVL C01738 V=800.0 PL=0
MOVL C01739 V=800.0 PL=0
MOVL C01740 V=800.0 PL=0
MOVL C01741 V=800.0 PL=0
MOVL C01742 V=800.0 PL=0
MOVL C01743 V=800.0 PL=0
MOVL C01744 V=800.0 PL=0
MOVL C01745 V=800.0 PL=0
MOVL C01746 V=800.0 PL=0
MOVL C01747 V=800.0 PL=0
MOVL C01748 V=800.0 PL=0
MOVL C01749 V=800.0 PL=0
MOVL C01750 V=800.0 PL=0
MOVL C01751 V=800.0 PL=0
MOVL C01752 V=800.0 PL=0
MOVL C01753 V=800.0 PL=0
MOVL C01754 V=800.0 PL=0
MOVL C01755 V=800.0 PL=0
MOVL C01756 V=800.0 PL=0
MOVL C01757 V=800.0 PL=0
MOVL C01758 V=800.0 PL=0
MOVL C01759 V=800.0 PL=0
MOVL C01760 V=800.0 PL=0
MOVL C01761 V=800.0 PL=0
MOVL C01762 V=800.0 PL=0
MOVL C01763 V=800.0 PL=0
MOVL C01764 V=800.0 PL=0
MOVL C01765 V=800.0 PL=0
MOVL C01766 V=800.0 PL=0
MOVL C01767 V=800.0 PL=0
MOVL C01768 V=800.0 PL=0
MOVL C01769 V=800.0 PL=0
MOVL C01770 V=800.0 PL=0
MOVL C01771 V=800.0 PL=0
MOVL C01772 V=800.0 PL=0
MOVL C01773 V=800.0 PL=0
MOVL C01774 V=800.0 PL=0
MOVL C01775 V=800.0 PL=0
MOVL C01776 V=800.0 PL=0
MOVL C01777 V=800.0 PL=0
MOVL C01778 V=800.0 PL=0
MOVL C01779 V=800.0 PL=0
MOVL C01780 V=800.0 PL=0
MOVL C01781 V=800.0 PL=0
MOVL C01782 V=800.0 PL=0
MOVL C01783 V=800.0 PL=0
MOVL C01784 V=800.0 PL=0
MOVL C01785 V=800.0 PL=0
MOVL C01786 V=800.0 PL=0
MOVL C01787 V=800.0 PL=0
MOVL C01788 V=800.0 PL=0
MOVL C01789 V=800.0 PL=0
MOVL C01790 V=800.0 PL=0
MOVL C01791 V=800.0 PL=0
MOVL C01792 V=800.0 PL=0
MOVL C01793 V=800.0 PL=0
MOVL C01794 V=800.0 PL=0
MOVL C01795 V=800.0 PL=0
MOVL C01796 V=800.0 PL=0
MOVL C01797 V=800.0 PL=0
MOVL C01798 V=800.0 PL=0
MOVL C01799 V=800.0 PL=0
MOVL C01800 V=800.0 PL=0
MOVL C01801 V=800.0 PL=0
MOVL C01802 V=800.0 PL=0
MOVL C01803 V=800.0 PL=0
MOVL C01804 V=800.0 PL=0
MOVL C01805 V=800.0 PL=0
MOVL C01806 V=800.0 PL=0
MOVL C01807 V=800.0 PL=0
MOVL C01808 V=800.0 PL=0
MOVL C01809 V=800.0 PL=0
MOVL C01810 V=800.0 PL=0
MOVL C01811 V=800.0 PL=0
MOVL C01812 V=800.0 PL=0
MOVL C01813 V=800.0 PL=0
MOVL C01814 V=800.0 PL=0
MOVL C01815 V=800.0 PL=0
MOVL C01816 V=800.0 PL=0
MOVL C01817 V=800.0 PL=0
MOVL C01818 V=800.0 PL=0
MOVL C01819 V=800.0 PL=0
MOVL C01820 V=800.0 PL=0
MOVL C01821 V=800.0 PL=0
MOVL C01822 V=800.0 PL=0
MOVL C01823 V=800.0 PL=0
MOVL C01824 V=800.0 PL=0
MOVL C01825 V=800.0 PL=0
MOVL C01826 V=800.0 PL=0
MOVL C01827 V=800.0 PL=0
MOVL C01828 V=800.0 PL=0
MOVL C01829 V=800.0 PL=0
MOVL C01830 V=800.0 PL=0
MOVL C01831 V=800.0 PL=0
MOVL C01832 V=800.0 PL=0
MOVL C01833 V=800.0 PL=0
MOVL C01834 V=800.0 PL=0
MOVL C01835 V=800.0 PL=0
MOVL C01836 V=800.0 PL=0
MOVL C01837 V=800.0 PL=0
MOVL C01838 V=800.0 PL=0
MOVL C01839 V=800.0 PL=0
MOVL C01840 V=800.0 PL=0
MOVL C01841 V=800.0 PL=0
MOVL C01842 V=800.0 PL=0
MOVL C01843 V=800.0 PL=0
MOVL C01844 V=800.0 PL=0
MOVL C01845 V=800.0 PL=0
MOVL C01846 V=800.0 PL=0
MOVL C01847 V=800.0 PL=0
MOVL C01848 V=800.0 PL=0
MOVL C01849 V=800.0 PL=0
MOVL C01850 V=800.0 PL=0
MOVL C01851 V=800.0 PL=0
MOVL C01852 V=800.0 PL=0
MOVL C01853 V=800.0 PL=0
MOVL C01854 V=800.0 PL=0
MOVL C01855 V=800.0 PL=0
MOVL C01856 V=800.0 PL=0
MOVL C01857 V=800.0 PL=0
MOVL C01858 V=800.0 PL=0
MOVL C01859 V=800.0 PL=0
MOVL C01860 V=800.0 PL=0
MOVL C01861 V=800.0 PL=0
MOVL C01862 V=800.0 PL=0
MOVL C01863 V=800.0 PL=0
MOVL C01864 V=800.0 PL=0
MOVL C01865 V=800.0 PL=0
MOVL C01866 V=800.0 PL=0
MOVL C01867 V=800.0 PL=0
MOVL C01868 V=800.0 PL=0
MOVL C01869 V=800.0 PL=0
MOVL C01870 V=800.0 PL=0
MOVL C01871 V=800.0 PL=0
MOVL C01872 V=800.0 PL=0
MOVL C01873 V=800.0 PL=0
MOVL C01874 V=800.0 PL=0
MOVL C01875 V=800.0 PL=0
MOVL C01876 V=800.0 PL=0
MOVL C01877 V=800.0 PL=0
MOVL C01878 V=800.0 PL=0
MOVL C01879 V=800.0 PL=0
MOVL C01880 V=800.0 PL=0
MOVL C01881 V=800.0 PL=0
MOVL C01882 V=800.0 PL=0
MOVL C01883 V=800.0 PL=0
MOVL C01884 V=800.0 PL=0
MOVL C01885 V=800.0 PL=0
MOVL C01886 V=800.0 PL=0
MOVL C01887 V=800.0 PL=0
MOVL C01888 V=800.0 PL=0
MOVL C01889 V=800.0 PL=0
MOVL C01890 V=800.0 PL=0
MOVL C01891 V=800.0 PL=0
MOVL C01892 V=800.0 PL=0
MOVL C01893 V=800.0 PL=0
MOVL C01894 V=800.0 PL=0
MOVL C01895 V=800.0 PL=0
MOVL C01896 V=800.0 PL=0
MOVL C01897 V=800.0 PL=0
MOVL C01898 V=800.0 PL=0
MOVL C01899 V=800.0 PL=0
MOVL C01900 V=800.0 PL=0
MOVL C01901 V=800.0 PL=0
MOVL C01902 V=800.0 PL=0
MOVL C01903 V=800.0 PL=0
MOVL C01904 V=800.0 PL=0
MOVL C01905 V=800.0 PL=0
MOVL C01906 V=800.0 PL=0
MOVL C01907 V=800.0 PL=0
MOVL C01908 V=800.0 PL=0
MOVL C01909 V=800.0 PL=0
MOVL C01910 V=800.0 PL=0
MOVL C01911 V=800.0 PL=0
MOVL C01912 V=800.0 PL=0
MOVL C01913 V=800.0 PL=0
MOVL C01914 V=800.0 PL=0
MOVL C01915 V=800.0 PL=0
MOVL C01916 V=800.0 PL=0
MOVL C01917 V=800.0 PL=0
MOVL C01918 V=800.0 PL=0
MOVL C01919 V=800.0 PL=0
MOVL C01920 V=800.0 PL=0
MOVL C01921 V=800.0 PL=0
MOVL C01922 V=800.0 PL=0
MOVL C01923 V=800.0 PL=0
MOVL C01924 V=800.0 PL=0
MOVL C01925 V=800.0 PL=0
MOVL C01926 V=800.0 PL=0
MOVL C01927 V=800.0 PL=0
MOVL C01928 V=800.0 PL=0
MOVL C01929 V=800.0 PL=0
MOVL C01930 V=800.0 PL=0
MOVL C01931 V=800.0 PL=0
MOVL C01932 V=800.0 PL=0
MOVL C01933 V=800.0 PL=0
MOVL C01934 V=800.0 PL=0
MOVL C01935 V=800.0 PL=0
MOVL C01936 V=800.0 PL=0
MOVL C01937 V=800.0 PL=0
MOVL C01938 V=800.0 PL=0
MOVL C01939 V=800.0 PL=0
MOVL C01940 V=800.0 PL=0
MOVL C01941 V=800.0 PL=0
MOVL C01942 V=800.0 PL=0
MOVL C01943 V=800.0 PL=0
MOVL C01944 V=800.0 PL=0
MOVL C01945 V=800.0 PL=0
MOVL C01946 V=800.0 PL=0
MOVL C01947 V=800.0 PL=0
MOVL C01948 V=800.0 PL=0
MOVL C01949 V=800.0 PL=0
MOVL C01950 V=800.0 PL=0
MOVL C01951 V=800.0 PL=0
MOVL C01952 V=800.0 PL=0
MOVL C01953 V=800.0 PL=0
MOVL C01954 V=800.0 PL=0
MOVL C01955 V=800.0 PL=0
MOVL C01956 V=800.0 PL=0
MOVL C01957 V=800.0 PL=0
MOVL C01958 V=800.0 PL=0
MOVL C01959 V=800.0 PL=0
MOVL C01960 V=800.0 PL=0
MOVL C01961 V=800.0 PL=0
MOVL C01962 V=800.0 PL=0
MOVL C01963 V=800.0 PL=0
MOVL C01964 V=800.0 PL=0
MOVL C01965 V=800.0 PL=0
MOVL C01966 V=800.0 PL=0
MOVL C01967 V=800.0 PL=0
MOVL C01968 V=800.0 PL=0
MOVL C01969 V=800.0 PL=0
MOVL C01970 V=800.0 PL=0
MOVL C01971 V=800.0 PL=0
MOVL C01972 V=800.0 PL=0
MOVL C01973 V=800.0 PL=0
MOVL C01974 V=800.0 PL=0
MOVL C01975 V=800.0 PL=0
MOVL C01976 V=800.0 PL=0
MOVL C01977 V=800.0 PL=0
MOVL C01978 V=800.0 PL=0
MOVL C01979 V=800.0 PL=0
MOVL C01980 V=800.0 PL=0
MOVL C01981 V=800.0 PL=0
MOVL C01982 V=800.0 PL=0
MOVL C01983 V=800.0 PL=0
MOVL C01984 V=800.0 PL=0
MOVL C01985 V=800.0 PL=0
MOVL C01986 V=800.0 PL=0
MOVL C01987 V=800.0 PL=0
MOVL C01988 V=800.0 PL=0
MOVL C01989 V=800.0 PL=0
MOVL C01990 V=800.0 PL=0
MOVL C01991 V=800.0 PL=0
MOVL C01992 V=800.0 PL=0
MOVL C01993 V=800.0 PL=0
MOVL C01994 V=800.0 PL=0
MOVL C01995 V=800.0 PL=0
MOVL C01996 V=800.0 PL=0
MOVL C01997 V=800.0 PL=0
MOVL C01998 V=800.0 PL=0
MOVL C01999 V=800.0 PL=0
MOVL C02000 V=800.0 PL=0
MOVL C02001 V=800.0 PL=0
MOVL C02002 V=800.0 PL=0
MOVL C02003 V=800.0 PL=0
MOVL C02004 V=800.0 PL=0
MOVL C02005 V=800.0 PL=0
MOVL C02006 V=800.0 PL=0
MOVL C02007 V=800.0 PL=0
MOVL C02008 V=800.0 PL=0
MOVL C02009 V=800.0 PL=0
MOVL C02010 V=800.0 PL=0
MOVL C02011 V=800.0 PL=0
MOVL C02012 V=800.0 PL=0
MOVL C02013 V=800.0 PL=0
MOVL C02014 V=800.0 PL=0
MOVL C02015 V=800.0 PL=0
MOVL C02016 V=800.0 PL=0
MOVL C02017 V=800.0 PL=0
MOVL C02018 V=800.0 PL=0
MOVL C02019 V=800.0 PL=0
MOVL C02020 V=800.0 PL=0
MOVL C02021 V=800.0 PL=0
MOVL C02022 V=800.0 PL=0
MOVL C02023 V=800.0 PL=0
MOVL C02024 V=800.0 PL=0
MOVL C02025 V=800.0 PL=0
MOVL C02026 V=800.0 PL=0
MOVL C02027 V=800.0 PL=0
MOVL C02028 V=800.0 PL=0
MOVL C02029 V=800.0 PL=0
MOVL C02030 V=800.0 PL=0
MOVL C02031 V=800.0 PL=0
MOVL C02032 V=800.0 PL=0
MOVL C02033 V=800.0 PL=0
MOVL C02034 V=800.0 PL=0
MOVL C02035 V=800.0 PL=0
MOVL C02036 V=800.0 PL=0
MOVL C02037 V=800.0 PL=0
MOVL C02038 V=800.0 PL=0
MOVL C02039 V=800.0 PL=0
MOVL C02040 V=800.0 PL=0
MOVL C02041 V=800.0 PL=0
MOVL C02042 V=800.0 PL=0
MOVL C02043 V=800.0 PL=0
MOVL C02044 V=800.0 PL=0
MOVL C02045 V=800.0 PL=0
MOVL C02046 V=800.0 PL=0
MOVL C02047 V=800.0 PL=0
MOVL C02048 V=800.0 PL=0
MOVL C02049 V=800.0 PL=0
MOVL C02050 V=800.0 PL=0
MOVL C02051 V=800.0 PL=0
MOVL C02052 V=800.0 PL=0
MOVL C02053 V=800.0 PL=0
MOVL C02054 V=800.0 PL=0
MOVL C02055 V=800.0 PL=0
MOVL C02056 V=800.0 PL=0
MOVL C02057 V=800.0 PL=0
MOVL C02058 V=800.0 PL=0
MOVL C02059 V=800.0 PL=0
MOVL C02060 V=800.0 PL=0
MOVL C02061 V=800.0 PL=0
MOVL C02062 V=800.0 PL=0
MOVL C02063 V=800.0 PL=0
MOVL C02064 V=800.0 PL=0
MOVL C02065 V=800.0 PL=0
MOVL C02066 V=800.0 PL=0
MOVL C02067 V=800.0 PL=0
MOVL C02068 V=800.0 PL=0
MOVL C02069 V=800.0 PL=0
MOVL C02070 V=800.0 PL=0
MOVL C02071 V=800.0 PL=0
MOVL C02072 V=800.0 PL=0
MOVL C02073 V=800.0 PL=0
MOVL C02074 V=800.0 PL=0
MOVL C02075 V=800.0 PL=0
MOVL C02076 V=800.0 PL=0
MOVL C02077 V=800.0 PL=0
MOVL C02078 V=800.0 PL=0
MOVL C02079 V=800.0 PL=0
MOVL C02080 V=800.0 PL=0
MOVL C02081 V=800.0 PL=0
MOVL C02082 V=800.0 PL=0
MOVL C02083 V=800.0 PL=0
MOVL C02084 V=800.0 PL=0
MOVL C02085 V=800.0 PL=0
MOVL C02086 V=800.0 PL=0
MOVL C02087 V=800.0 PL=0
MOVL C02088 V=800.0 PL=0
MOVL C02089 V=800.0 PL=0
MOVL C02090 V=800.0 PL=0
MOVL C02091 V=800.0 PL=0
MOVL C02092 V=800.0 PL=0
MOVL C02093 V=800.0 PL=0
MOVL C02094 V=800.0 PL=0
MOVL C02095 V=800.0 PL=0
MOVL C02096 V=800.0 PL=0
MOVL C02097 V=800.0 PL=0
MOVL C02098 V=800.0 PL=0
MOVL C02099 V=800.0 PL=0
MOVL C02100 V=800.0 PL=0
MOVL C02101 V=800.0 PL=0
MOVL C02102 V=800.0 PL=0
MOVL C02103 V=800.0 PL=0
MOVL C02104 V=800.0 PL=0
MOVL C02105 V=800.0 PL=0
MOVL C02106 V=800.0 PL=0
MOVL C02107 V=800.0 PL=0
MOVL C02108 V=800.0 PL=0
MOVL C02109 V=800.0 PL=0
MOVL C02110 V=800.0 PL=0
MOVL C02111 V=800.0 PL=0
MOVL C02112 V=800.0 PL=0
MOVL C02113 V=800.0 PL=0
MOVL C02114 V=800.0 PL=0
MOVL C02115 V=800.0 PL=0
MOVL C02116 V=800.0 PL=0
MOVL C02117 V=800.0 PL=0
MOVL C02118 V=800.0 PL=0
